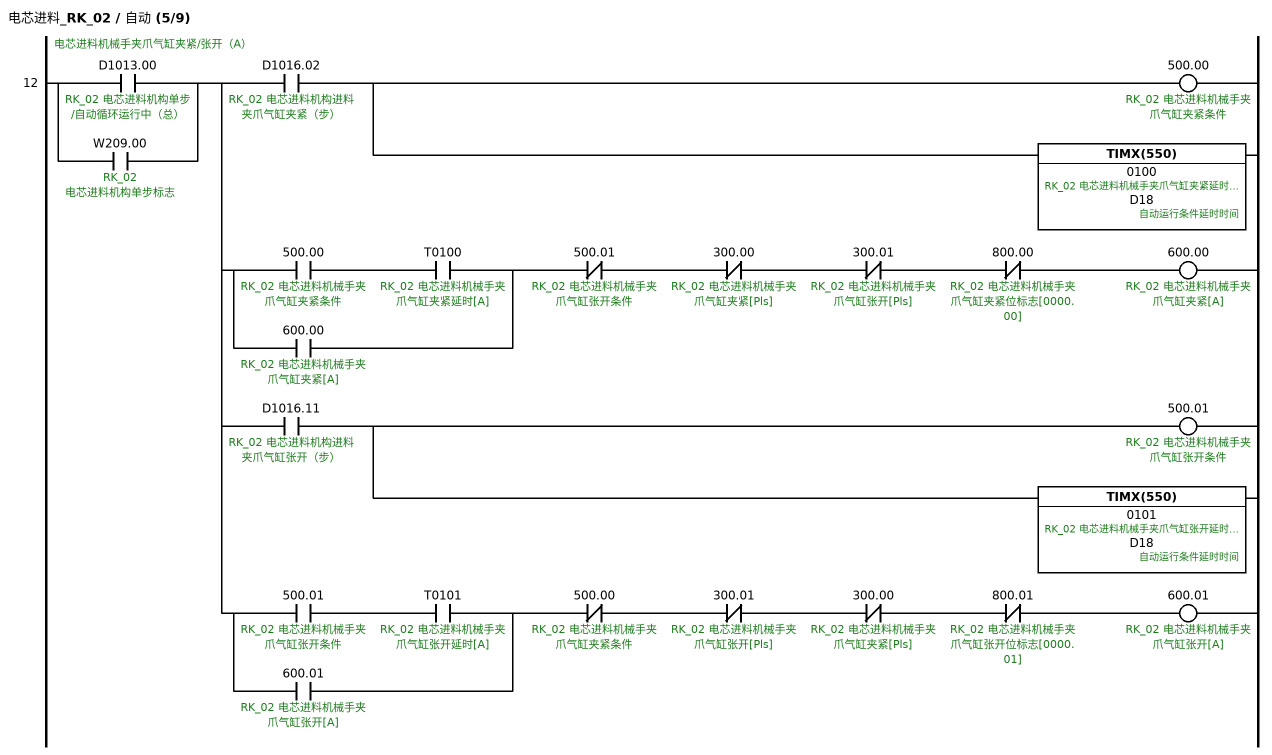
; [picture p360: 电芯进料_RK_02 / 自动, rungs 12-12]
; rung 12: 电芯进料机械手夹爪气缸夹紧/张开（A）
LD D1013.00  ; RK_02 电芯进料机构单步/自动循环运行中（总）
OR W209.00  ; RK_02  电芯进料机构单步标志
OUT TR0
AND D1016.02  ; RK_02 电芯进料机构进料夹爪气缸夹紧（步）
OUT 500.00  ; RK_02 电芯进料机械手夹爪气缸夹紧条件
TIMX(550) 0100 D18  ; 自动运行条件延时时间, RK_02 电芯进料机械手夹爪气缸夹紧延时[A]
LD TR0
LD 500.00  ; RK_02 电芯进料机械手夹爪气缸夹紧条件
AND T0100  ; RK_02 电芯进料机械手夹爪气缸夹紧延时[A]
OR 600.00  ; RK_02 电芯进料机械手夹爪气缸夹紧[A]
ANDLD
ANDNOT 500.01  ; RK_02 电芯进料机械手夹爪气缸张开条件
ANDNOT 300.00  ; RK_02 电芯进料机械手夹爪气缸夹紧[Pls]
ANDNOT 300.01  ; RK_02 电芯进料机械手夹爪气缸张开[Pls]
ANDNOT 800.00  ; RK_02 电芯进料机械手夹爪气缸夹紧位标志[0000.00]
OUT 600.00  ; RK_02 电芯进料机械手夹爪气缸夹紧[A]
LD TR0
AND D1016.11  ; RK_02 电芯进料机构进料夹爪气缸张开（步）
OUT 500.01  ; RK_02 电芯进料机械手夹爪气缸张开条件
TIMX(550) 0101 D18  ; 自动运行条件延时时间, RK_02 电芯进料机械手夹爪气缸张开延时[A]
LD TR0
LD 500.01  ; RK_02 电芯进料机械手夹爪气缸张开条件
AND T0101  ; RK_02 电芯进料机械手夹爪气缸张开延时[A]
OR 600.01  ; RK_02 电芯进料机械手夹爪气缸张开[A]
ANDLD
ANDNOT 500.00  ; RK_02 电芯进料机械手夹爪气缸夹紧条件
ANDNOT 300.01  ; RK_02 电芯进料机械手夹爪气缸张开[Pls]
ANDNOT 300.00  ; RK_02 电芯进料机械手夹爪气缸夹紧[Pls]
ANDNOT 800.01  ; RK_02 电芯进料机械手夹爪气缸张开位标志[0000.01]
OUT 600.01  ; RK_02 电芯进料机械手夹爪气缸张开[A]

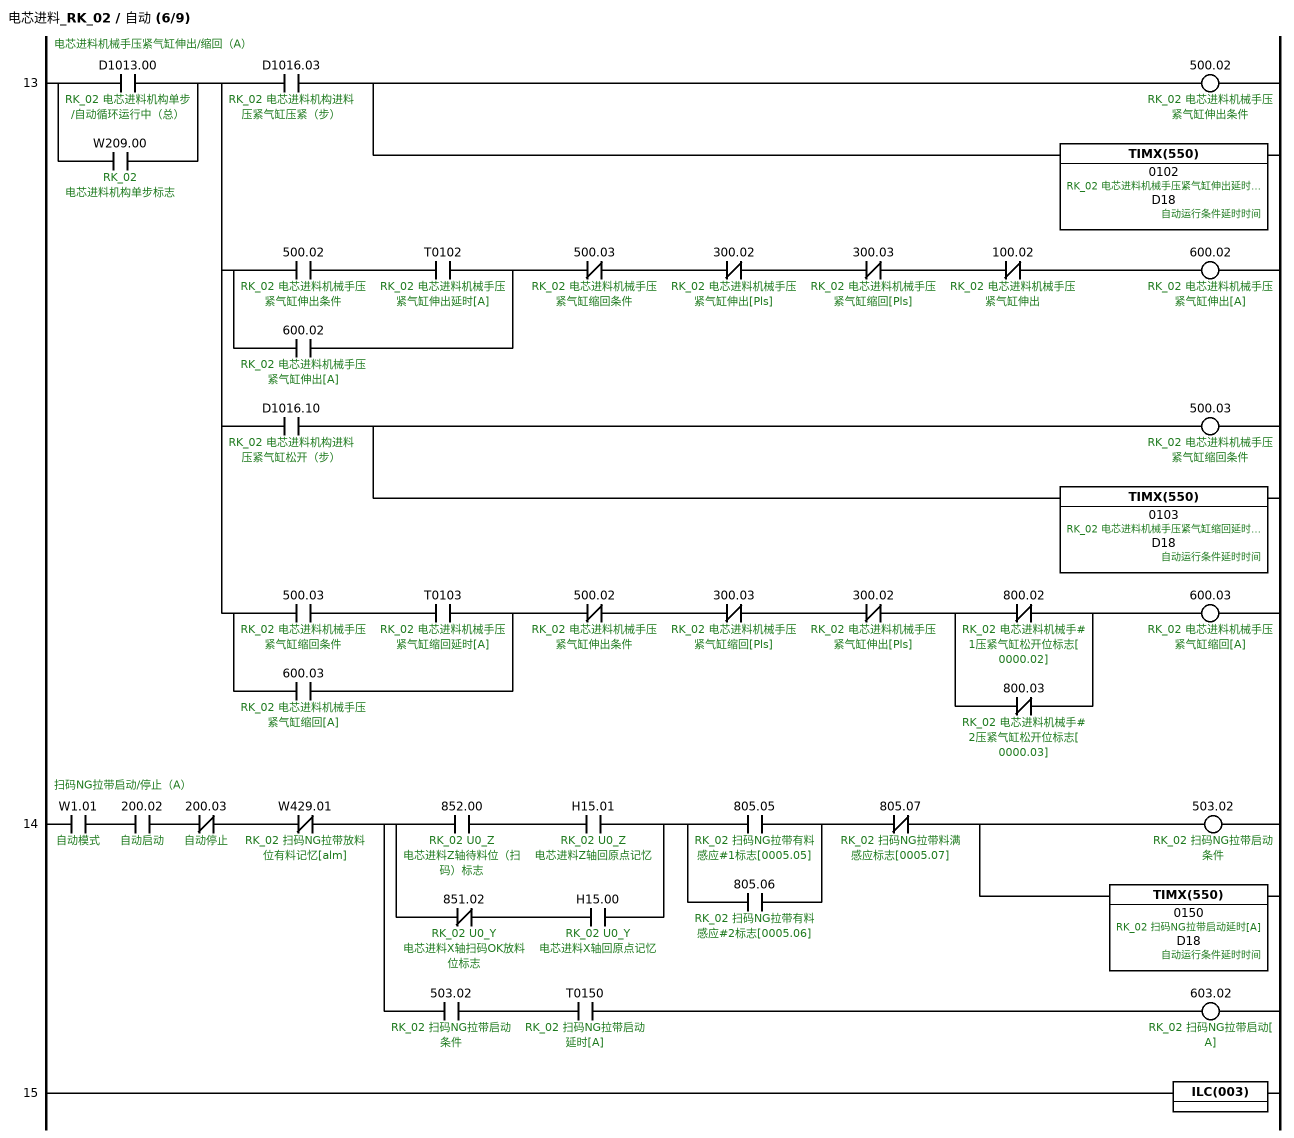
; rung 13: 电芯进料机械手压紧气缸伸出/缩回（A）
LD D1013.00  ; RK_02 电芯进料机构单步/自动循环运行中（总）
OR W209.00  ; RK_02  电芯进料机构单步标志
OUT TR0
AND D1016.03  ; RK_02 电芯进料机构进料压紧气缸压紧（步）
OUT 500.02  ; RK_02 电芯进料机械手压紧气缸伸出条件
TIMX(550) 0102 D18  ; 自动运行条件延时时间, RK_02 电芯进料机械手压紧气缸伸出延时[A]
LD TR0
LD 500.02  ; RK_02 电芯进料机械手压紧气缸伸出条件
AND T0102  ; RK_02 电芯进料机械手压紧气缸伸出延时[A]
OR 600.02  ; RK_02 电芯进料机械手压紧气缸伸出[A]
ANDLD
ANDNOT 500.03  ; RK_02 电芯进料机械手压紧气缸缩回条件
ANDNOT 300.02  ; RK_02 电芯进料机械手压紧气缸伸出[Pls]
ANDNOT 300.03  ; RK_02 电芯进料机械手压紧气缸缩回[Pls]
ANDNOT 100.02  ; RK_02 电芯进料机械手压紧气缸伸出
OUT 600.02  ; RK_02 电芯进料机械手压紧气缸伸出[A]
LD TR0
AND D1016.10  ; RK_02 电芯进料机构进料压紧气缸松开（步）
OUT 500.03  ; RK_02 电芯进料机械手压紧气缸缩回条件
TIMX(550) 0103 D18  ; 自动运行条件延时时间, RK_02 电芯进料机械手压紧气缸缩回延时[A]
LD TR0
LD 500.03  ; RK_02 电芯进料机械手压紧气缸缩回条件
AND T0103  ; RK_02 电芯进料机械手压紧气缸缩回延时[A]
OR 600.03  ; RK_02 电芯进料机械手压紧气缸缩回[A]
ANDLD
ANDNOT 500.02  ; RK_02 电芯进料机械手压紧气缸伸出条件
ANDNOT 300.03  ; RK_02 电芯进料机械手压紧气缸缩回[Pls]
ANDNOT 300.02  ; RK_02 电芯进料机械手压紧气缸伸出[Pls]
LDNOT 800.02  ; RK_02 电芯进料机械手#1压紧气缸松开位标志[0000.02]
ORNOT 800.03  ; RK_02 电芯进料机械手#2压紧气缸松开位标志[0000.03]
ANDLD
OUT 600.03  ; RK_02 电芯进料机械手压紧气缸缩回[A]
; rung 14: 扫码NG拉带启动/停止（A）
LD W1.01  ; 自动模式
AND 200.02  ; 自动启动
ANDNOT 200.03  ; 自动停止
ANDNOT W429.01  ; RK_02 扫码NG拉带放料位有料记忆[alm]
OUT TR0
LD 852.00  ; RK_02 U0_Z 电芯进料Z轴待料位（扫码）标志
AND H15.01  ; RK_02 U0_Z 电芯进料Z轴回原点记忆
LDNOT 851.02  ; RK_02 U0_Y 电芯进料X轴扫码OK放料位标志
AND H15.00  ; RK_02 U0_Y 电芯进料X轴回原点记忆
ORLD
ANDLD
LD 805.05  ; RK_02 扫码NG拉带有料感应#1标志[0005.05]
OR 805.06  ; RK_02 扫码NG拉带有料感应#2标志[0005.06]
ANDLD
ANDNOT 805.07  ; RK_02 扫码NG拉带料满感应标志[0005.07]
OUT 503.02  ; RK_02 扫码NG拉带启动条件
TIMX(550) 0150 D18  ; 自动运行条件延时时间, RK_02 扫码NG拉带启动延时[A]
LD TR0
AND 503.02  ; RK_02 扫码NG拉带启动条件
AND T0150  ; RK_02 扫码NG拉带启动延时[A]
OUT 603.02  ; RK_02 扫码NG拉带启动[A]
; rung 15
ILC(003)

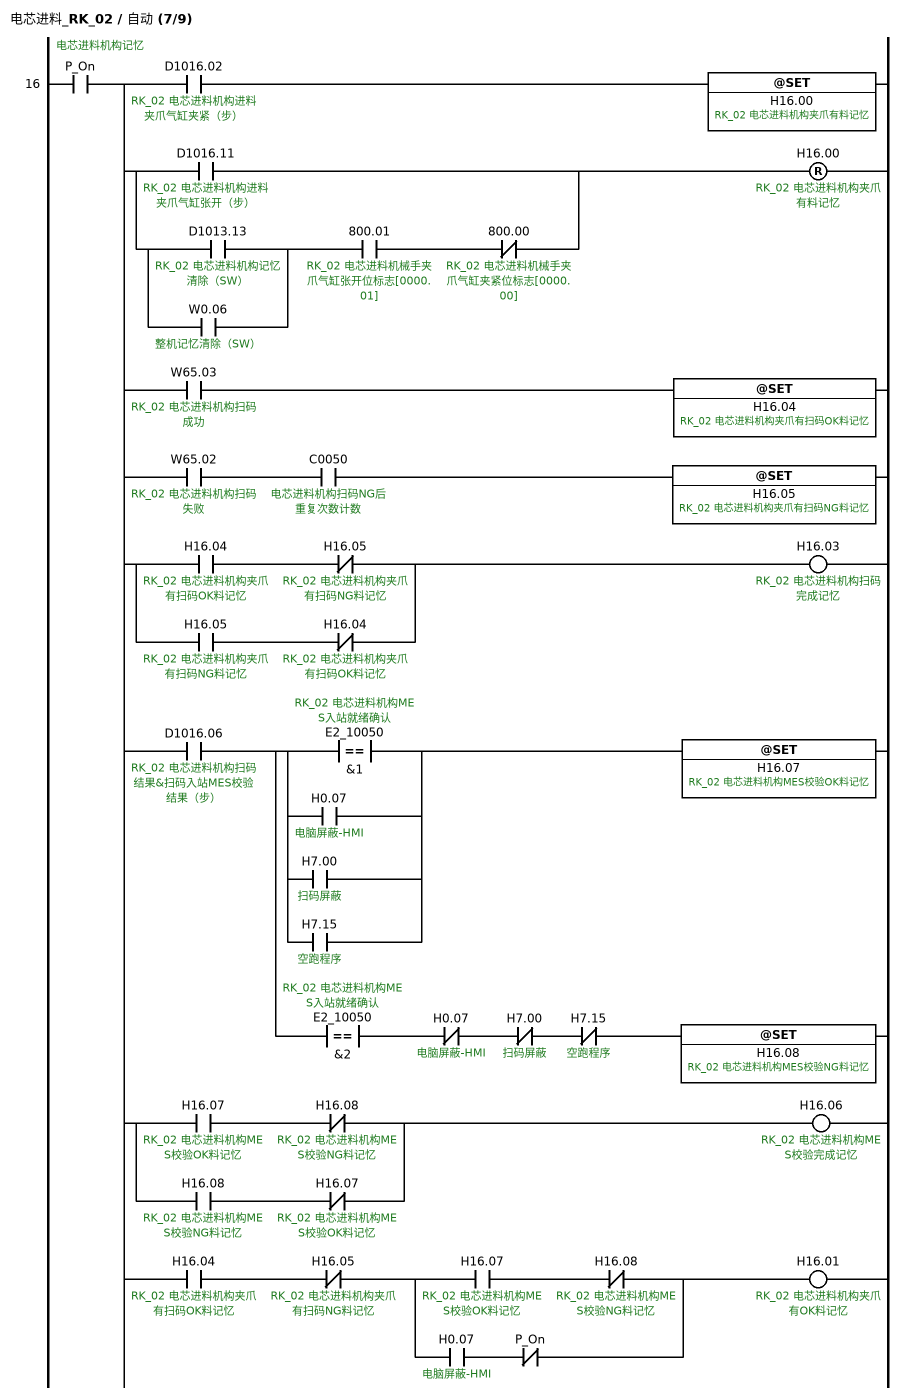

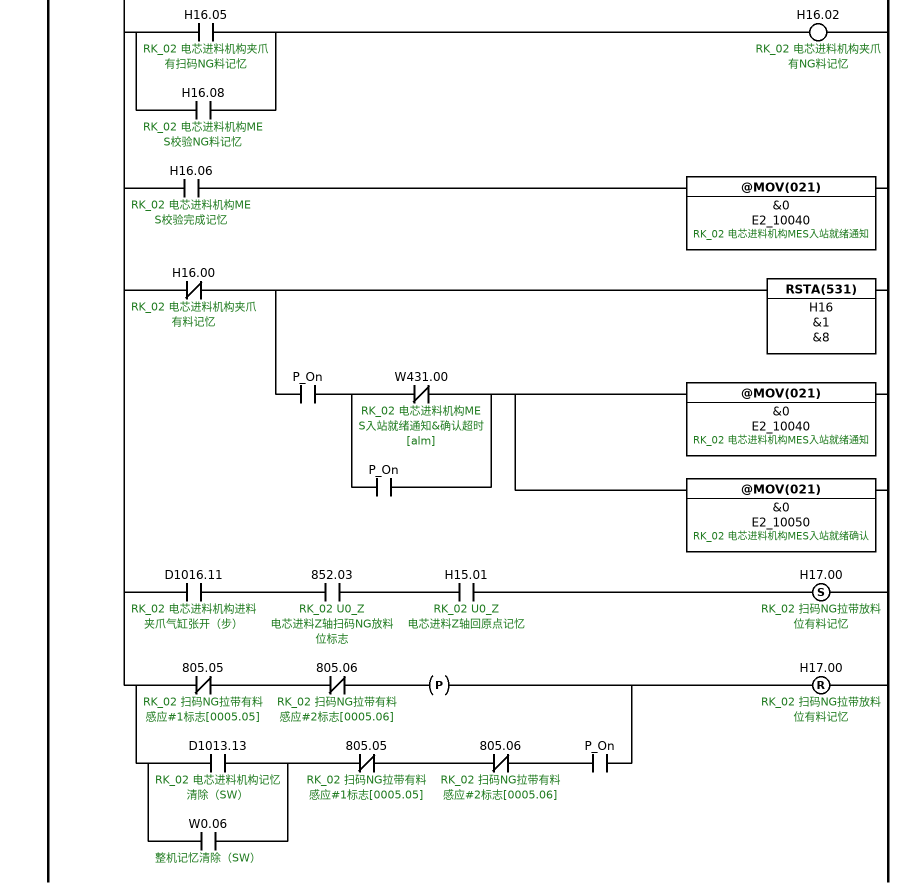
; rung 16: 电芯进料机构记忆
LD P_On
OUT TR0
AND D1016.02  ; RK_02 电芯进料机构进料夹爪气缸夹紧（步）
@SET H16.00  ; RK_02 电芯进料机构夹爪有料记忆
LD TR0
LD D1016.11  ; RK_02 电芯进料机构进料夹爪气缸张开（步）
LD D1013.13  ; RK_02 电芯进料机构记忆清除（SW）
OR W0.06  ; 整机记忆清除（SW）
AND 800.01  ; RK_02 电芯进料机械手夹爪气缸张开位标志[0000.01]
ANDNOT 800.00  ; RK_02 电芯进料机械手夹爪气缸夹紧位标志[0000.00]
ORLD
ANDLD
RSET H16.00  ; RK_02 电芯进料机构夹爪有料记忆
LD TR0
AND W65.03  ; RK_02 电芯进料机构扫码成功
@SET H16.04  ; RK_02 电芯进料机构夹爪有扫码OK料记忆
LD TR0
AND W65.02  ; RK_02 电芯进料机构扫码失败
AND C0050  ; 电芯进料机构扫码NG后重复次数计数
@SET H16.05  ; RK_02 电芯进料机构夹爪有扫码NG料记忆
LD TR0
LD H16.04  ; RK_02 电芯进料机构夹爪有扫码OK料记忆
ANDNOT H16.05  ; RK_02 电芯进料机构夹爪有扫码NG料记忆
LD H16.05  ; RK_02 电芯进料机构夹爪有扫码NG料记忆
ANDNOT H16.04  ; RK_02 电芯进料机构夹爪有扫码OK料记忆
ORLD
ANDLD
OUT H16.03  ; RK_02 电芯进料机构扫码完成记忆
LD TR0
AND D1016.06  ; RK_02 电芯进料机构扫码结果&扫码入站MES校验结果（步）
OUT TR1
LD=(300) E2_10050 &1  ; RK_02 电芯进料机构MES入站就绪确认  // 入站就绪确认=0：未确认，1：确认OK，2：确认NG
OR H0.07  ; 电脑屏蔽-HMI
OR H7.00  ; 扫码屏蔽
OR H7.15  ; 空跑程序
ANDLD
@SET H16.07  ; RK_02 电芯进料机构MES校验OK料记忆
LD TR1
AND=(300) E2_10050 &2  ; RK_02 电芯进料机构MES入站就绪确认  // 入站就绪确认=0：未确认，1：确认OK，2：确认NG
ANDNOT H0.07  ; 电脑屏蔽-HMI
ANDNOT H7.00  ; 扫码屏蔽
ANDNOT H7.15  ; 空跑程序
@SET H16.08  ; RK_02 电芯进料机构MES校验NG料记忆
LD TR0
LD H16.07  ; RK_02 电芯进料机构MES校验OK料记忆
ANDNOT H16.08  ; RK_02 电芯进料机构MES校验NG料记忆
LD H16.08  ; RK_02 电芯进料机构MES校验NG料记忆
ANDNOT H16.07  ; RK_02 电芯进料机构MES校验OK料记忆
ORLD
ANDLD
OUT H16.06  ; RK_02 电芯进料机构MES校验完成记忆
LD TR0
AND H16.04  ; RK_02 电芯进料机构夹爪有扫码OK料记忆
ANDNOT H16.05  ; RK_02 电芯进料机构夹爪有扫码NG料记忆
LD H16.07  ; RK_02 电芯进料机构MES校验OK料记忆
ANDNOT H16.08  ; RK_02 电芯进料机构MES校验NG料记忆
LD H0.07  ; 电脑屏蔽-HMI
ANDNOT P_On
ORLD
ANDLD
OUT H16.01  ; RK_02 电芯进料机构夹爪有OK料记忆
LD TR0
LD H16.05  ; RK_02 电芯进料机构夹爪有扫码NG料记忆
OR H16.08  ; RK_02 电芯进料机构MES校验NG料记忆
ANDLD
OUT H16.02  ; RK_02 电芯进料机构夹爪有NG料记忆
LD TR0
AND H16.06  ; RK_02 电芯进料机构MES校验完成记忆
@MOV(021) &0 E2_10040  ; RK_02 电芯进料机构MES入站就绪通知
LD TR0
ANDNOT H16.00  ; RK_02 电芯进料机构夹爪有料记忆
RSTA(531) H16 &1 &8
AND P_On
LDNOT W431.00  ; RK_02 电芯进料机构MES入站就绪通知&确认超时[alm]  // 工站夹爪没料且无MES入站就绪通知&确认报警条件下，RK_02 电芯进料机构MES入站就绪通知&确认才能清零
OR P_On
ANDLD
@MOV(021) &0 E2_10040  ; RK_02 电芯进料机构MES入站就绪通知
@MOV(021) &0 E2_10050  ; RK_02 电芯进料机构MES入站就绪确认
LD TR0
AND D1016.11  ; RK_02 电芯进料机构进料夹爪气缸张开（步）
AND 852.03  ; RK_02 U0_Z 电芯进料Z轴扫码NG放料位标志
AND H15.01  ; RK_02 U0_Z 电芯进料Z轴回原点记忆
SET H17.00  ; RK_02 扫码NG拉带放料位有料记忆
LD TR0
LDNOT 805.05  ; RK_02 扫码NG拉带有料感应#1标志[0005.05]
ANDNOT 805.06  ; RK_02 扫码NG拉带有料感应#2标志[0005.06]
UP(521)
LD D1013.13  ; RK_02 电芯进料机构记忆清除（SW）
OR W0.06  ; 整机记忆清除（SW）
ANDNOT 805.05  ; RK_02 扫码NG拉带有料感应#1标志[0005.05]
ANDNOT 805.06  ; RK_02 扫码NG拉带有料感应#2标志[0005.06]
AND P_On
ORLD
ANDLD
RSET H17.00  ; RK_02 扫码NG拉带放料位有料记忆

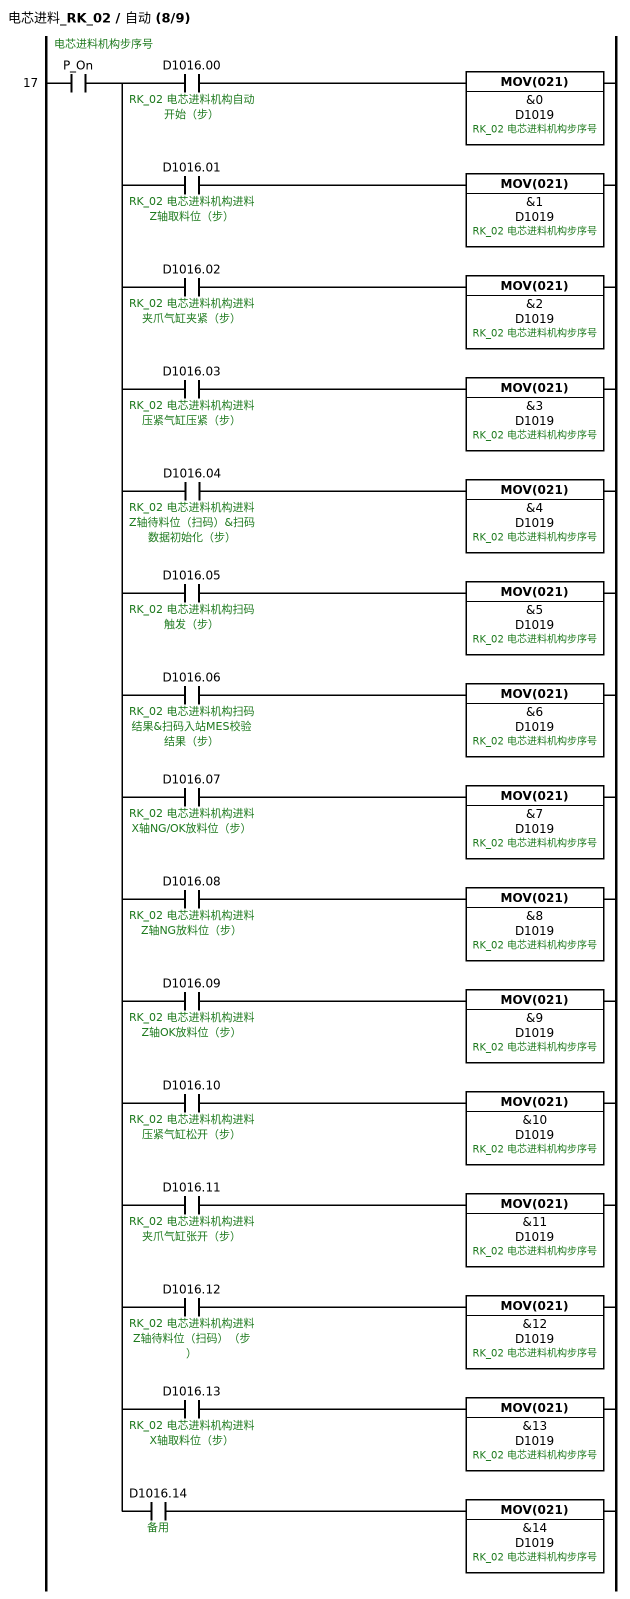
; rung 17: 电芯进料机构步序号
LD P_On
OUT TR0
AND D1016.00  ; RK_02 电芯进料机构自动开始（步）
MOV(021) &0 D1019  ; RK_02 电芯进料机构步序号
LD TR0
AND D1016.01  ; RK_02 电芯进料机构进料Z轴取料位（步）
MOV(021) &1 D1019  ; RK_02 电芯进料机构步序号
LD TR0
AND D1016.02  ; RK_02 电芯进料机构进料夹爪气缸夹紧（步）
MOV(021) &2 D1019  ; RK_02 电芯进料机构步序号
LD TR0
AND D1016.03  ; RK_02 电芯进料机构进料压紧气缸压紧（步）
MOV(021) &3 D1019  ; RK_02 电芯进料机构步序号
LD TR0
AND D1016.04  ; RK_02 电芯进料机构进料Z轴待料位（扫码）&扫码数据初始化（步）
MOV(021) &4 D1019  ; RK_02 电芯进料机构步序号
LD TR0
AND D1016.05  ; RK_02 电芯进料机构扫码触发（步）
MOV(021) &5 D1019  ; RK_02 电芯进料机构步序号
LD TR0
AND D1016.06  ; RK_02 电芯进料机构扫码结果&扫码入站MES校验结果（步）
MOV(021) &6 D1019  ; RK_02 电芯进料机构步序号
LD TR0
AND D1016.07  ; RK_02 电芯进料机构进料X轴NG/OK放料位（步）
MOV(021) &7 D1019  ; RK_02 电芯进料机构步序号
LD TR0
AND D1016.08  ; RK_02 电芯进料机构进料Z轴NG放料位（步）
MOV(021) &8 D1019  ; RK_02 电芯进料机构步序号
LD TR0
AND D1016.09  ; RK_02 电芯进料机构进料Z轴OK放料位（步）
MOV(021) &9 D1019  ; RK_02 电芯进料机构步序号
LD TR0
AND D1016.10  ; RK_02 电芯进料机构进料压紧气缸松开（步）
MOV(021) &10 D1019  ; RK_02 电芯进料机构步序号
LD TR0
AND D1016.11  ; RK_02 电芯进料机构进料夹爪气缸张开（步）
MOV(021) &11 D1019  ; RK_02 电芯进料机构步序号
LD TR0
AND D1016.12  ; RK_02 电芯进料机构进料Z轴待料位（扫码）（步）
MOV(021) &12 D1019  ; RK_02 电芯进料机构步序号
LD TR0
AND D1016.13  ; RK_02 电芯进料机构进料X轴取料位（步）
MOV(021) &13 D1019  ; RK_02 电芯进料机构步序号
LD TR0
AND D1016.14  ; 备用
MOV(021) &14 D1019  ; RK_02 电芯进料机构步序号

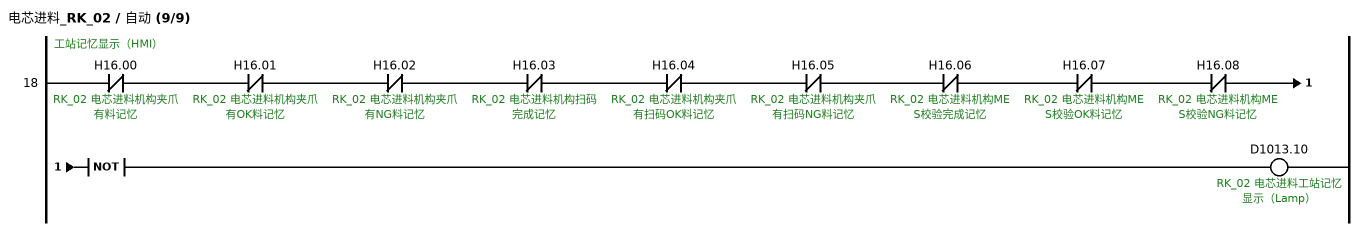
; rung 18: 工站记忆显示（HMI）
LDNOT H16.00  ; RK_02 电芯进料机构夹爪有料记忆
ANDNOT H16.01  ; RK_02 电芯进料机构夹爪有OK料记忆
ANDNOT H16.02  ; RK_02 电芯进料机构夹爪有NG料记忆
ANDNOT H16.03  ; RK_02 电芯进料机构扫码完成记忆
ANDNOT H16.04  ; RK_02 电芯进料机构夹爪有扫码OK料记忆
ANDNOT H16.05  ; RK_02 电芯进料机构夹爪有扫码NG料记忆
ANDNOT H16.06  ; RK_02 电芯进料机构MES校验完成记忆
ANDNOT H16.07  ; RK_02 电芯进料机构MES校验OK料记忆
ANDNOT H16.08  ; RK_02 电芯进料机构MES校验NG料记忆
NOT(520)
OUT D1013.10  ; RK_02 电芯进料工站记忆显示（Lamp）

### Section 复位

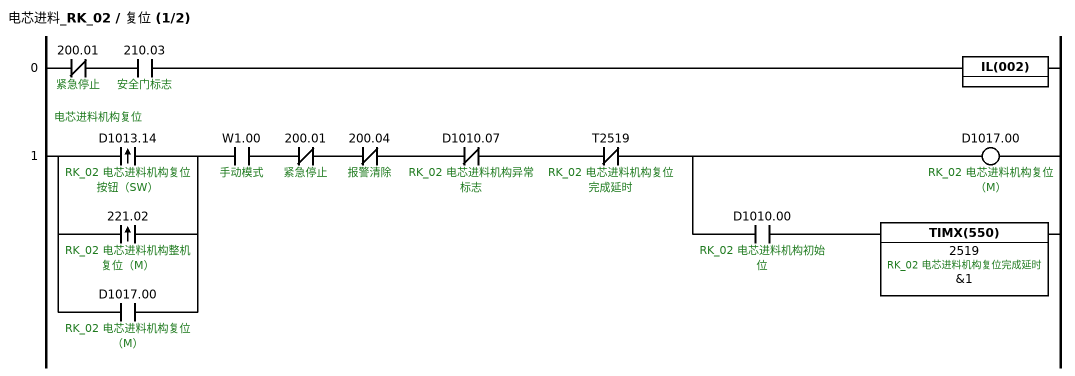
; rung 0
LDNOT 200.01  ; 紧急停止
AND 210.03  ; 安全门标志
IL(002)
; rung 1: 电芯进料机构复位
@LD D1013.14  ; RK_02 电芯进料机构复位按钮（SW）
@OR 221.02  ; RK_02 电芯进料机构整机复位（M）
OR D1017.00  ; RK_02 电芯进料机构复位（M）
AND W1.00  ; 手动模式
ANDNOT 200.01  ; 紧急停止
ANDNOT 200.04  ; 报警清除
ANDNOT D1010.07  ; RK_02 电芯进料机构异常标志
ANDNOT T2519  ; RK_02 电芯进料机构复位完成延时
OUT D1017.00  ; RK_02 电芯进料机构复位（M）
AND D1010.00  ; RK_02 电芯进料机构初始位
TIMX(550) 2519 &1  ; RK_02 电芯进料机构复位完成延时

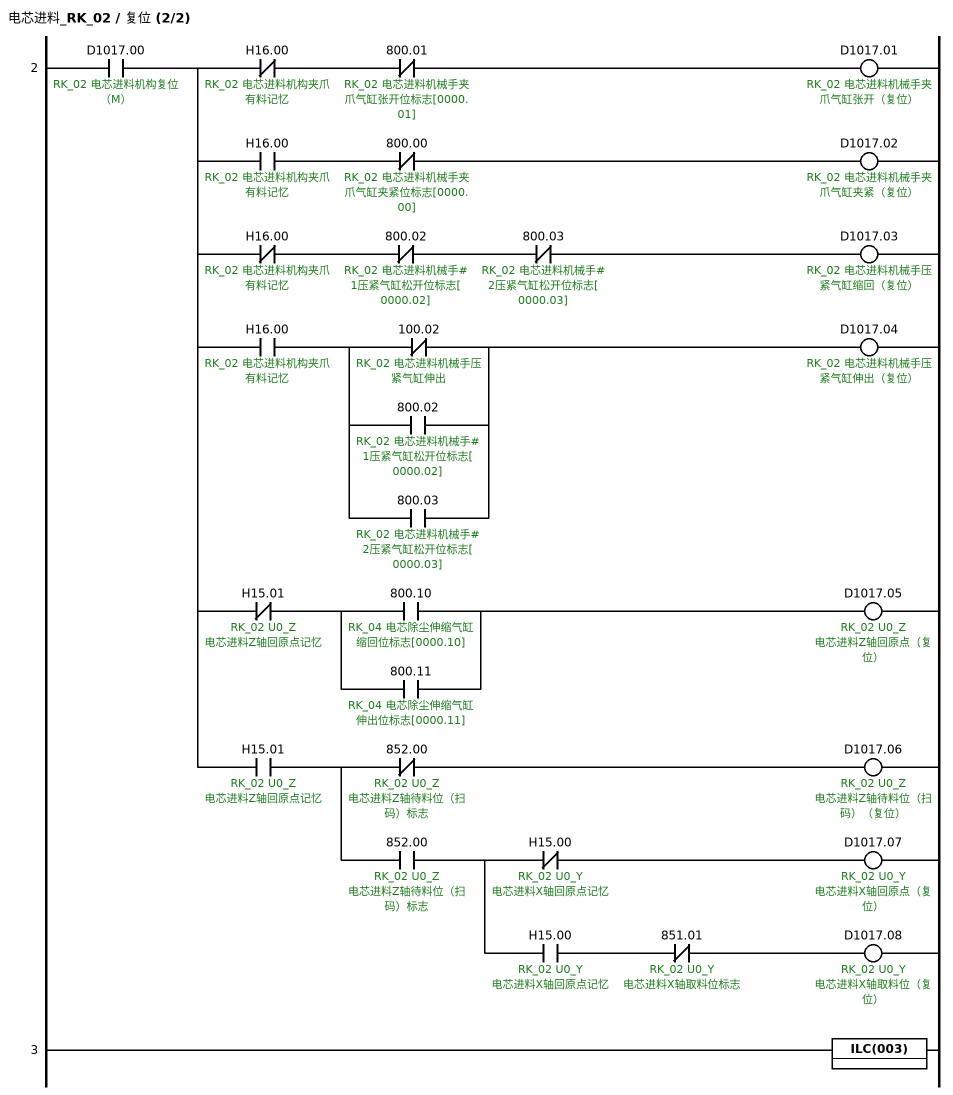
; rung 2
LD D1017.00  ; RK_02 电芯进料机构复位（M）
OUT TR0
ANDNOT H16.00  ; RK_02 电芯进料机构夹爪有料记忆
ANDNOT 800.01  ; RK_02 电芯进料机械手夹爪气缸张开位标志[0000.01]
OUT D1017.01  ; RK_02 电芯进料机械手夹爪气缸张开（复位）
LD TR0
AND H16.00  ; RK_02 电芯进料机构夹爪有料记忆
ANDNOT 800.00  ; RK_02 电芯进料机械手夹爪气缸夹紧位标志[0000.00]
OUT D1017.02  ; RK_02 电芯进料机械手夹爪气缸夹紧（复位）
LD TR0
ANDNOT H16.00  ; RK_02 电芯进料机构夹爪有料记忆
ANDNOT 800.02  ; RK_02 电芯进料机械手#1压紧气缸松开位标志[0000.02]
ANDNOT 800.03  ; RK_02 电芯进料机械手#2压紧气缸松开位标志[0000.03]
OUT D1017.03  ; RK_02 电芯进料机械手压紧气缸缩回（复位）
LD TR0
AND H16.00  ; RK_02 电芯进料机构夹爪有料记忆
LDNOT 100.02  ; RK_02 电芯进料机械手压紧气缸伸出
OR 800.02  ; RK_02 电芯进料机械手#1压紧气缸松开位标志[0000.02]
OR 800.03  ; RK_02 电芯进料机械手#2压紧气缸松开位标志[0000.03]
ANDLD
OUT D1017.04  ; RK_02 电芯进料机械手压紧气缸伸出（复位）
LD TR0
ANDNOT H15.01  ; RK_02 U0_Z 电芯进料Z轴回原点记忆
LD 800.10  ; RK_04 电芯除尘伸缩气缸缩回位标志[0000.10]
OR 800.11  ; RK_04 电芯除尘伸缩气缸伸出位标志[0000.11]
ANDLD
OUT D1017.05  ; RK_02 U0_Z 电芯进料Z轴回原点（复位）
LD TR0
AND H15.01  ; RK_02 U0_Z 电芯进料Z轴回原点记忆
OUT TR0
ANDNOT 852.00  ; RK_02 U0_Z 电芯进料Z轴待料位（扫码）标志
OUT D1017.06  ; RK_02 U0_Z 电芯进料Z轴待料位（扫码）（复位）
LD TR0
AND 852.00  ; RK_02 U0_Z 电芯进料Z轴待料位（扫码）标志
OUT TR0
ANDNOT H15.00  ; RK_02 U0_Y 电芯进料X轴回原点记忆
OUT D1017.07  ; RK_02 U0_Y 电芯进料X轴回原点（复位）
LD TR0
AND H15.00  ; RK_02 U0_Y 电芯进料X轴回原点记忆
ANDNOT 851.01  ; RK_02 U0_Y 电芯进料X轴取料位标志
OUT D1017.08  ; RK_02 U0_Y 电芯进料X轴取料位（复位）
; rung 3
ILC(003)

### Section 指示灯

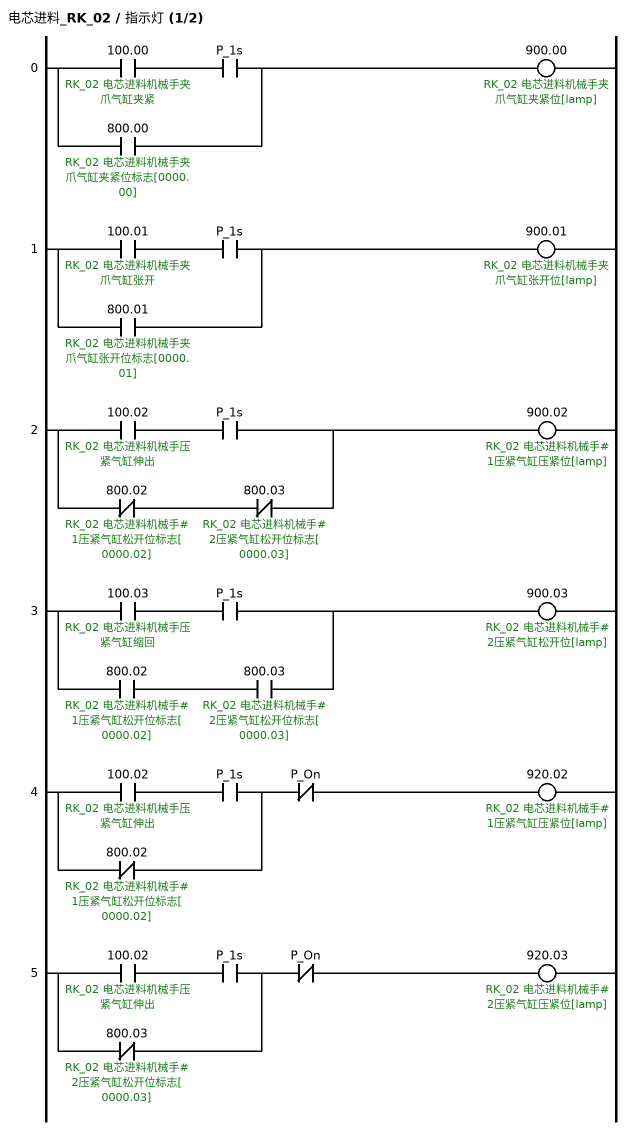
; rung 0
LD 100.00  ; RK_02 电芯进料机械手夹爪气缸夹紧
AND P_1s
OR 800.00  ; RK_02 电芯进料机械手夹爪气缸夹紧位标志[0000.00]
OUT 900.00  ; RK_02 电芯进料机械手夹爪气缸夹紧位[lamp]
; rung 1
LD 100.01  ; RK_02 电芯进料机械手夹爪气缸张开
AND P_1s
OR 800.01  ; RK_02 电芯进料机械手夹爪气缸张开位标志[0000.01]
OUT 900.01  ; RK_02 电芯进料机械手夹爪气缸张开位[lamp]
; rung 2
LD 100.02  ; RK_02 电芯进料机械手压紧气缸伸出
AND P_1s
LDNOT 800.02  ; RK_02 电芯进料机械手#1压紧气缸松开位标志[0000.02]
ANDNOT 800.03  ; RK_02 电芯进料机械手#2压紧气缸松开位标志[0000.03]
ORLD
OUT 900.02  ; RK_02 电芯进料机械手#1压紧气缸压紧位[lamp]
; rung 3
LD 100.03  ; RK_02 电芯进料机械手压紧气缸缩回
AND P_1s
LD 800.02  ; RK_02 电芯进料机械手#1压紧气缸松开位标志[0000.02]
AND 800.03  ; RK_02 电芯进料机械手#2压紧气缸松开位标志[0000.03]
ORLD
OUT 900.03  ; RK_02 电芯进料机械手#2压紧气缸松开位[lamp]
; rung 4
LD 100.02  ; RK_02 电芯进料机械手压紧气缸伸出
AND P_1s
ORNOT 800.02  ; RK_02 电芯进料机械手#1压紧气缸松开位标志[0000.02]
ANDNOT P_On
OUT 920.02  ; RK_02 电芯进料机械手#1压紧气缸压紧位[lamp]
; rung 5
LD 100.02  ; RK_02 电芯进料机械手压紧气缸伸出
AND P_1s
ORNOT 800.03  ; RK_02 电芯进料机械手#2压紧气缸松开位标志[0000.03]
ANDNOT P_On
OUT 920.03  ; RK_02 电芯进料机械手#2压紧气缸压紧位[lamp]

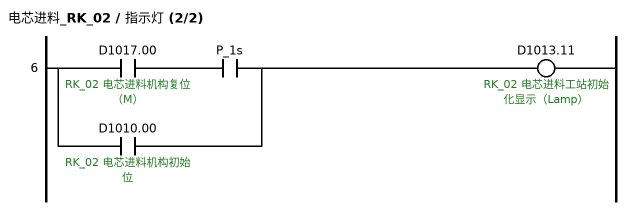
; rung 6
LD D1017.00  ; RK_02 电芯进料机构复位（M）
AND P_1s
OR D1010.00  ; RK_02 电芯进料机构初始位
OUT D1013.11  ; RK_02 电芯进料工站初始化显示（Lamp）

### Section 外部输出

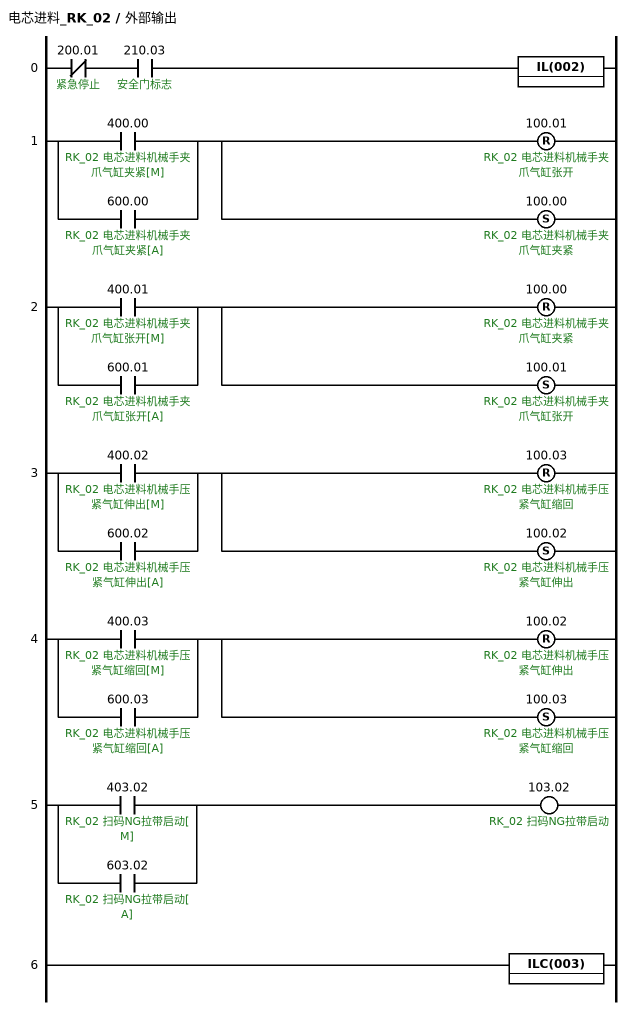
; rung 0
LDNOT 200.01  ; 紧急停止
AND 210.03  ; 安全门标志
IL(002)
; rung 1
LD 400.00  ; RK_02 电芯进料机械手夹爪气缸夹紧[M]
OR 600.00  ; RK_02 电芯进料机械手夹爪气缸夹紧[A]
RSET 100.01  ; RK_02 电芯进料机械手夹爪气缸张开
SET 100.00  ; RK_02 电芯进料机械手夹爪气缸夹紧
; rung 2
LD 400.01  ; RK_02 电芯进料机械手夹爪气缸张开[M]
OR 600.01  ; RK_02 电芯进料机械手夹爪气缸张开[A]
RSET 100.00  ; RK_02 电芯进料机械手夹爪气缸夹紧
SET 100.01  ; RK_02 电芯进料机械手夹爪气缸张开
; rung 3
LD 400.02  ; RK_02 电芯进料机械手压紧气缸伸出[M]
OR 600.02  ; RK_02 电芯进料机械手压紧气缸伸出[A]
RSET 100.03  ; RK_02 电芯进料机械手压紧气缸缩回
SET 100.02  ; RK_02 电芯进料机械手压紧气缸伸出
; rung 4
LD 400.03  ; RK_02 电芯进料机械手压紧气缸缩回[M]
OR 600.03  ; RK_02 电芯进料机械手压紧气缸缩回[A]
RSET 100.02  ; RK_02 电芯进料机械手压紧气缸伸出
SET 100.03  ; RK_02 电芯进料机械手压紧气缸缩回
; rung 5
LD 403.02  ; RK_02 扫码NG拉带启动[M]
OR 603.02  ; RK_02 扫码NG拉带启动[A]
OUT 103.02  ; RK_02 扫码NG拉带启动
; rung 6
ILC(003)

### Section END
; rung 0
END(001)

## Program 电芯上料_RK_03 (cyclic task 3)

### Section Main

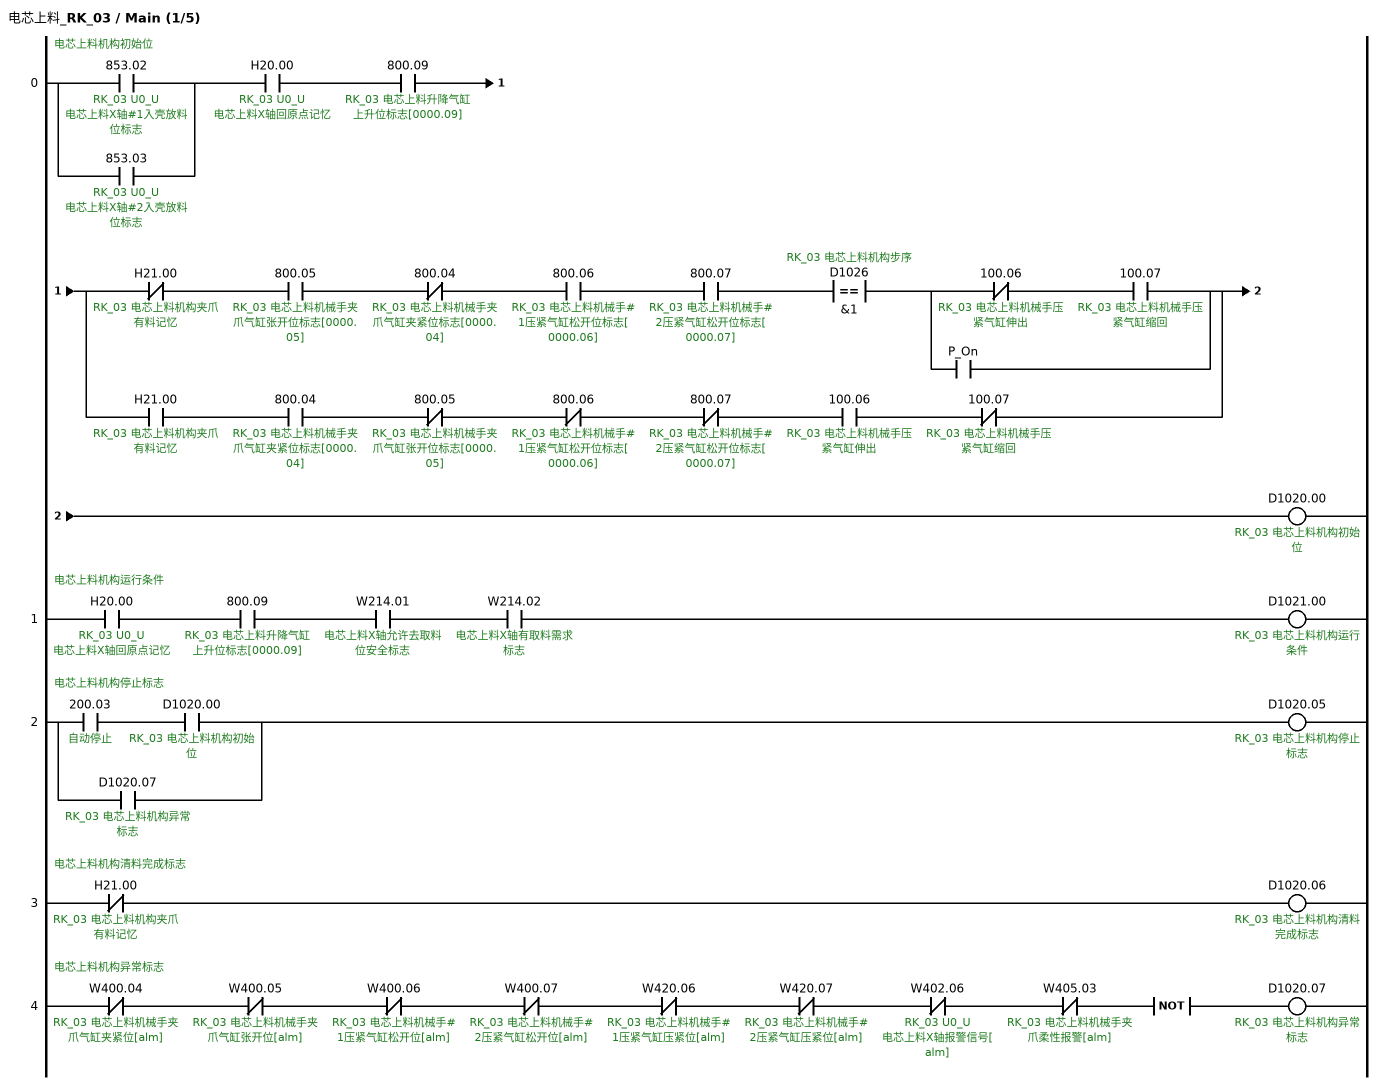
; rung 0: 电芯上料机构初始位
LD 853.02  ; RK_03 U0_U 电芯上料X轴#1入壳放料位标志
OR 853.03  ; RK_03 U0_U 电芯上料X轴#2入壳放料位标志
AND H20.00  ; RK_03 U0_U 电芯上料X轴回原点记忆
AND 800.09  ; RK_03 电芯上料升降气缸上升位标志[0000.09]
LDNOT H21.00  ; RK_03 电芯上料机构夹爪有料记忆
AND 800.05  ; RK_03 电芯上料机械手夹爪气缸张开位标志[0000.05]
ANDNOT 800.04  ; RK_03 电芯上料机械手夹爪气缸夹紧位标志[0000.04]
AND 800.06  ; RK_03 电芯上料机械手#1压紧气缸松开位标志[0000.06]
AND 800.07  ; RK_03 电芯上料机械手#2压紧气缸松开位标志[0000.07]
AND=(300) D1026 &1  ; RK_03 电芯上料机构步序
LDNOT 100.06  ; RK_03 电芯上料机械手压紧气缸伸出
AND 100.07  ; RK_03 电芯上料机械手压紧气缸缩回
OR P_On
ANDLD
LD H21.00  ; RK_03 电芯上料机构夹爪有料记忆
AND 800.04  ; RK_03 电芯上料机械手夹爪气缸夹紧位标志[0000.04]
ANDNOT 800.05  ; RK_03 电芯上料机械手夹爪气缸张开位标志[0000.05]
ANDNOT 800.06  ; RK_03 电芯上料机械手#1压紧气缸松开位标志[0000.06]
ANDNOT 800.07  ; RK_03 电芯上料机械手#2压紧气缸松开位标志[0000.07]
AND 100.06  ; RK_03 电芯上料机械手压紧气缸伸出
ANDNOT 100.07  ; RK_03 电芯上料机械手压紧气缸缩回
ORLD
ANDLD
OUT D1020.00  ; RK_03 电芯上料机构初始位
; rung 1: 电芯上料机构运行条件
LD H20.00  ; RK_03 U0_U 电芯上料X轴回原点记忆
AND 800.09  ; RK_03 电芯上料升降气缸上升位标志[0000.09]
AND W214.01  ; 电芯上料X轴允许去取料位安全标志
AND W214.02  ; 电芯上料X轴有取料需求标志
OUT D1021.00  ; RK_03 电芯上料机构运行条件
; rung 2: 电芯上料机构停止标志
LD 200.03  ; 自动停止
AND D1020.00  ; RK_03 电芯上料机构初始位
OR D1020.07  ; RK_03 电芯上料机构异常标志
OUT D1020.05  ; RK_03 电芯上料机构停止标志
; rung 3: 电芯上料机构清料完成标志
LDNOT H21.00  ; RK_03 电芯上料机构夹爪有料记忆
OUT D1020.06  ; RK_03 电芯上料机构清料完成标志
; rung 4: 电芯上料机构异常标志
LDNOT W400.04  ; RK_03 电芯上料机械手夹爪气缸夹紧位[alm]
ANDNOT W400.05  ; RK_03 电芯上料机械手夹爪气缸张开位[alm]
ANDNOT W400.06  ; RK_03 电芯上料机械手#1压紧气缸松开位[alm]
ANDNOT W400.07  ; RK_03 电芯上料机械手#2压紧气缸松开位[alm]
ANDNOT W420.06  ; RK_03 电芯上料机械手#1压紧气缸压紧位[alm]
ANDNOT W420.07  ; RK_03 电芯上料机械手#2压紧气缸压紧位[alm]
ANDNOT W402.06  ; RK_03 U0_U 电芯上料X轴报警信号[alm]
ANDNOT W405.03  ; RK_03 电芯上料机械手夹爪柔性报警[alm]
NOT(520)
OUT D1020.07  ; RK_03 电芯上料机构异常标志

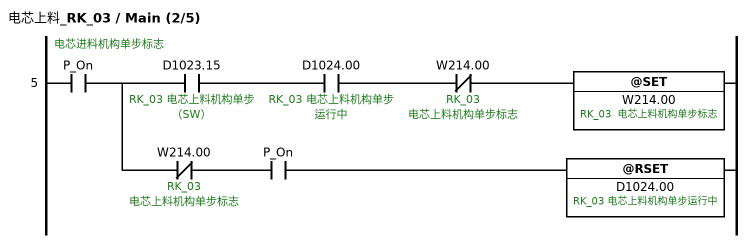
; rung 5: 电芯进料机构单步标志
LD P_On
OUT TR0
AND D1023.15  ; RK_03 电芯上料机构单步（SW）
AND D1024.00  ; RK_03 电芯上料机构单步运行中
ANDNOT W214.00  ; RK_03  电芯上料机构单步标志
@SET W214.00  ; RK_03  电芯上料机构单步标志
LD TR0
ANDNOT W214.00  ; RK_03  电芯上料机构单步标志
AND P_On
@RSET D1024.00  ; RK_03 电芯上料机构单步运行中

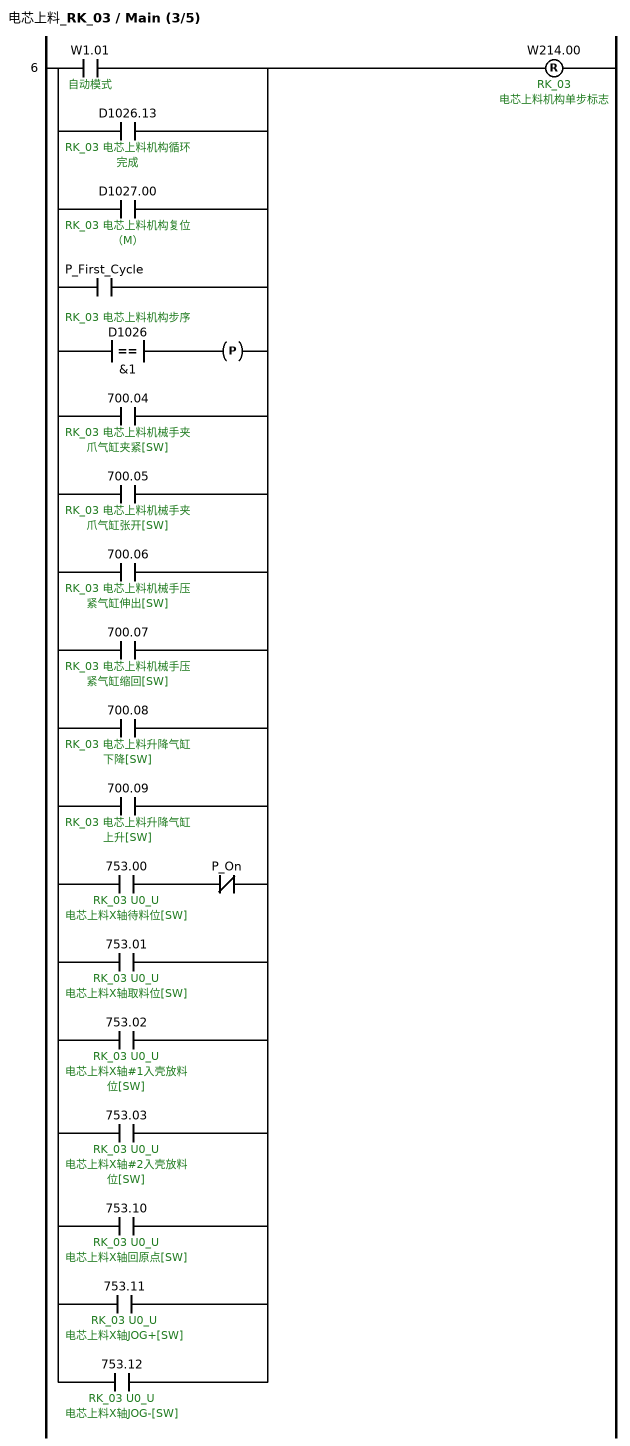
; rung 6
LD W1.01  ; 自动模式
OR D1026.13  ; RK_03 电芯上料机构循环完成
OR D1027.00  ; RK_03 电芯上料机构复位（M）
OR P_First_Cycle
LD=(300) D1026 &1  ; RK_03 电芯上料机构步序
UP(521)
ORLD
OR 700.04  ; RK_03 电芯上料机械手夹爪气缸夹紧[SW]
OR 700.05  ; RK_03 电芯上料机械手夹爪气缸张开[SW]
OR 700.06  ; RK_03 电芯上料机械手压紧气缸伸出[SW]
OR 700.07  ; RK_03 电芯上料机械手压紧气缸缩回[SW]
OR 700.08  ; RK_03 电芯上料升降气缸下降[SW]
OR 700.09  ; RK_03 电芯上料升降气缸上升[SW]
LD 753.00  ; RK_03 U0_U 电芯上料X轴待料位[SW]
ANDNOT P_On
ORLD
OR 753.01  ; RK_03 U0_U 电芯上料X轴取料位[SW]
OR 753.02  ; RK_03 U0_U 电芯上料X轴#1入壳放料位[SW]
OR 753.03  ; RK_03 U0_U 电芯上料X轴#2入壳放料位[SW]
OR 753.10  ; RK_03 U0_U 电芯上料X轴回原点[SW]
OR 753.11  ; RK_03 U0_U 电芯上料X轴JOG+[SW]
OR 753.12  ; RK_03 U0_U 电芯上料X轴JOG-[SW]
RSET W214.00  ; RK_03  电芯上料机构单步标志

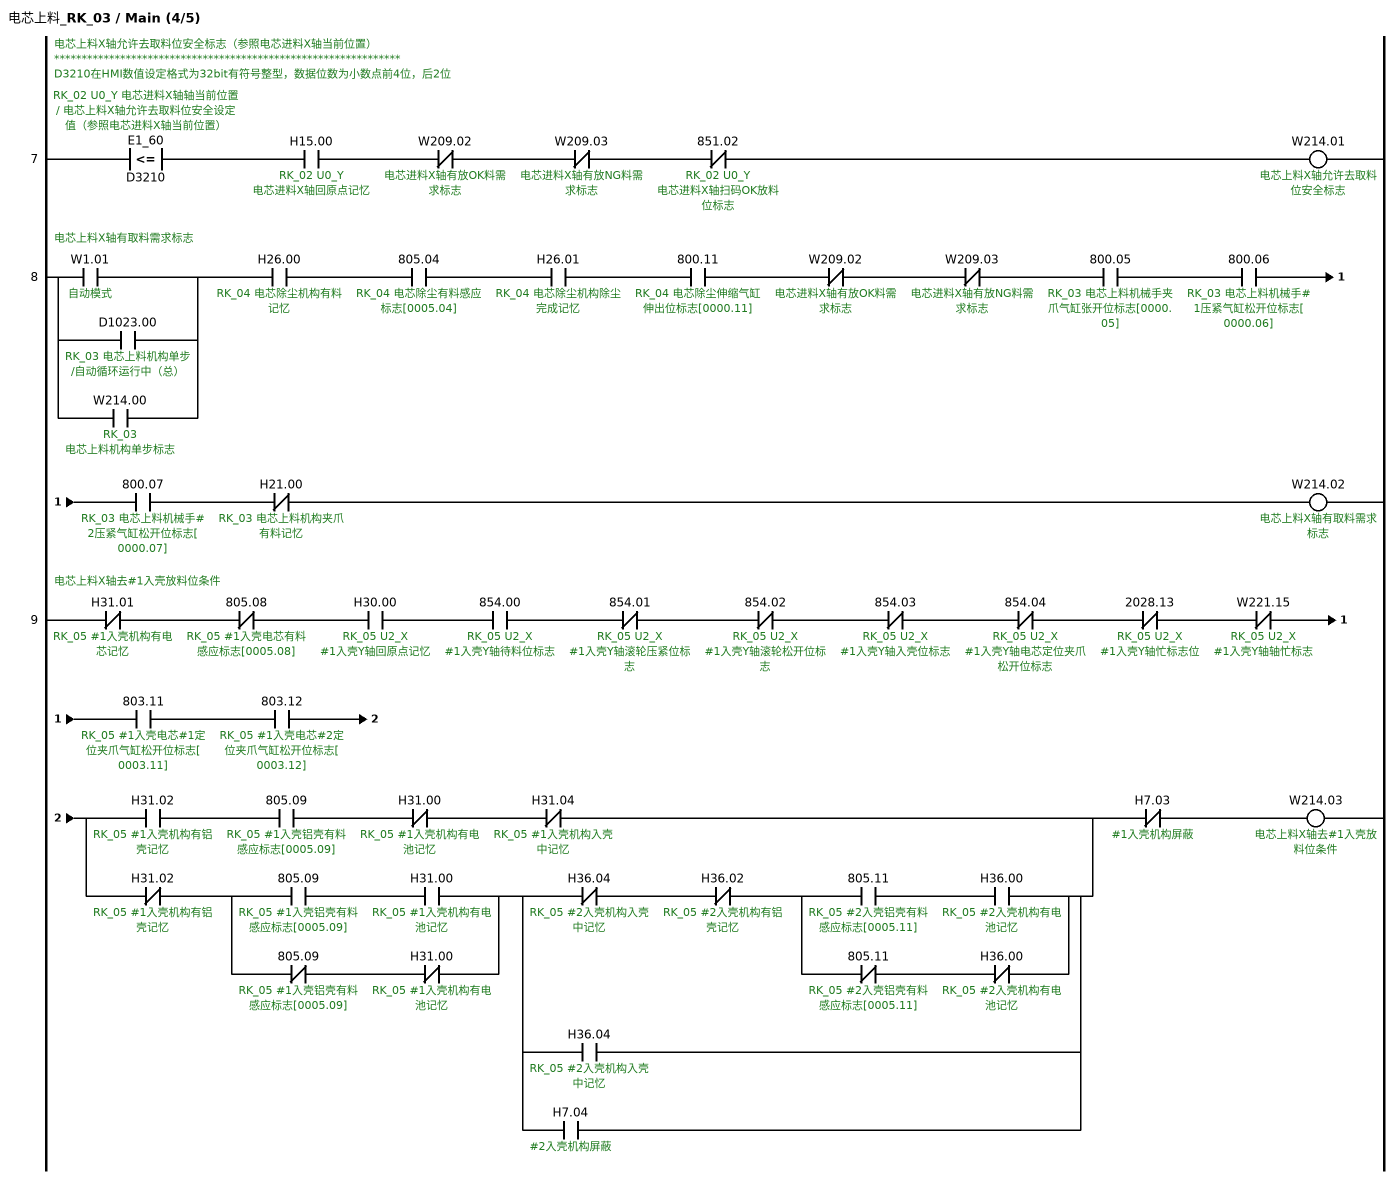
; rung 7: 电芯上料X轴允许去取料位安全标志（参照电芯进料X轴当前位置） / *************************************************************** / D3210在HMI数值设定格式为32bit有符号整型，数据位数为小数点前4位，后2位
LD<=SL(318) E1_60 D3210  ; RK_02 U0_Y 电芯进料X轴轴当前位置, 电芯上料X轴允许去取料位安全设定值（参照电芯进料X轴当前位置）
AND H15.00  ; RK_02 U0_Y 电芯进料X轴回原点记忆
ANDNOT W209.02  ; 电芯进料X轴有放OK料需求标志
ANDNOT W209.03  ; 电芯进料X轴有放NG料需求标志
ANDNOT 851.02  ; RK_02 U0_Y 电芯进料X轴扫码OK放料位标志
OUT W214.01  ; 电芯上料X轴允许去取料位安全标志
; rung 8: 电芯上料X轴有取料需求标志
LD W1.01  ; 自动模式
OR D1023.00  ; RK_03 电芯上料机构单步/自动循环运行中（总）
OR W214.00  ; RK_03  电芯上料机构单步标志
AND H26.00  ; RK_04 电芯除尘机构有料记忆
AND 805.04  ; RK_04 电芯除尘有料感应标志[0005.04]
AND H26.01  ; RK_04 电芯除尘机构除尘完成记忆
AND 800.11  ; RK_04 电芯除尘伸缩气缸伸出位标志[0000.11]
ANDNOT W209.02  ; 电芯进料X轴有放OK料需求标志
ANDNOT W209.03  ; 电芯进料X轴有放NG料需求标志
AND 800.05  ; RK_03 电芯上料机械手夹爪气缸张开位标志[0000.05]
AND 800.06  ; RK_03 电芯上料机械手#1压紧气缸松开位标志[0000.06]
AND 800.07  ; RK_03 电芯上料机械手#2压紧气缸松开位标志[0000.07]
ANDNOT H21.00  ; RK_03 电芯上料机构夹爪有料记忆
OUT W214.02  ; 电芯上料X轴有取料需求标志
; rung 9: 电芯上料X轴去#1入壳放料位条件
LDNOT H31.01  ; RK_05 #1入壳机构有电芯记忆
ANDNOT 805.08  ; RK_05 #1入壳电芯有料感应标志[0005.08]
AND H30.00  ; RK_05 U2_X #1入壳Y轴回原点记忆
AND 854.00  ; RK_05 U2_X #1入壳Y轴待料位标志
ANDNOT 854.01  ; RK_05 U2_X #1入壳Y轴滚轮压紧位标志
ANDNOT 854.02  ; RK_05 U2_X #1入壳Y轴滚轮松开位标志
ANDNOT 854.03  ; RK_05 U2_X #1入壳Y轴入壳位标志
ANDNOT 854.04  ; RK_05 U2_X #1入壳Y轴电芯定位夹爪松开位标志
ANDNOT 2028.13  ; RK_05 U2_X #1入壳Y轴忙标志位
ANDNOT W221.15  ; RK_05 U2_X #1入壳Y轴轴忙标志
AND 803.11  ; RK_05 #1入壳电芯#1定位夹爪气缸松开位标志[0003.11]
AND 803.12  ; RK_05 #1入壳电芯#2定位夹爪气缸松开位标志[0003.12]
LD H31.02  ; RK_05 #1入壳机构有铝壳记忆
AND 805.09  ; RK_05 #1入壳铝壳有料感应标志[0005.09]
ANDNOT H31.00  ; RK_05 #1入壳机构有电池记忆
ANDNOT H31.04  ; RK_05 #1入壳机构入壳中记忆
LDNOT H31.02  ; RK_05 #1入壳机构有铝壳记忆
LD 805.09  ; RK_05 #1入壳铝壳有料感应标志[0005.09]
AND H31.00  ; RK_05 #1入壳机构有电池记忆
LDNOT 805.09  ; RK_05 #1入壳铝壳有料感应标志[0005.09]
ANDNOT H31.00  ; RK_05 #1入壳机构有电池记忆
ORLD
ANDLD
LDNOT H36.04  ; RK_05 #2入壳机构入壳中记忆
ANDNOT H36.02  ; RK_05 #2入壳机构有铝壳记忆
LD 805.11  ; RK_05 #2入壳铝壳有料感应标志[0005.11]
AND H36.00  ; RK_05 #2入壳机构有电池记忆
LDNOT 805.11  ; RK_05 #2入壳铝壳有料感应标志[0005.11]
ANDNOT H36.00  ; RK_05 #2入壳机构有电池记忆
ORLD
ANDLD
OR H36.04  ; RK_05 #2入壳机构入壳中记忆
OR H7.04  ; #2入壳机构屏蔽
ANDLD
ORLD
ANDLD
ANDNOT H7.03  ; #1入壳机构屏蔽
OUT W214.03  ; 电芯上料X轴去#1入壳放料位条件

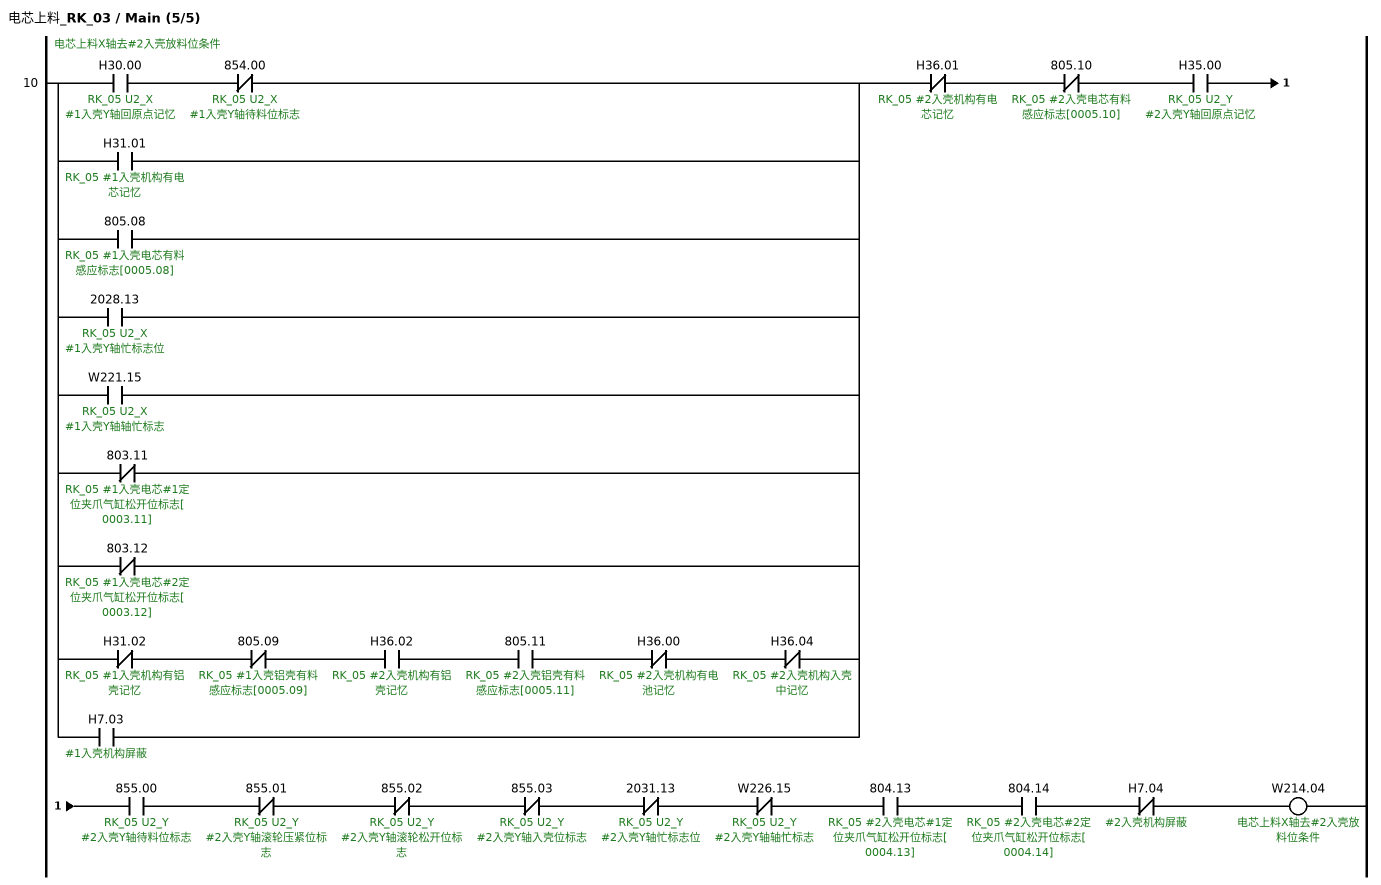
; rung 10: 电芯上料X轴去#2入壳放料位条件
LD H30.00  ; RK_05 U2_X #1入壳Y轴回原点记忆
ANDNOT 854.00  ; RK_05 U2_X #1入壳Y轴待料位标志
OR H31.01  ; RK_05 #1入壳机构有电芯记忆
OR 805.08  ; RK_05 #1入壳电芯有料感应标志[0005.08]
OR 2028.13  ; RK_05 U2_X #1入壳Y轴忙标志位
OR W221.15  ; RK_05 U2_X #1入壳Y轴轴忙标志
ORNOT 803.11  ; RK_05 #1入壳电芯#1定位夹爪气缸松开位标志[0003.11]
ORNOT 803.12  ; RK_05 #1入壳电芯#2定位夹爪气缸松开位标志[0003.12]
LDNOT H31.02  ; RK_05 #1入壳机构有铝壳记忆
ANDNOT 805.09  ; RK_05 #1入壳铝壳有料感应标志[0005.09]
AND H36.02  ; RK_05 #2入壳机构有铝壳记忆
AND 805.11  ; RK_05 #2入壳铝壳有料感应标志[0005.11]
ANDNOT H36.00  ; RK_05 #2入壳机构有电池记忆
ANDNOT H36.04  ; RK_05 #2入壳机构入壳中记忆
ORLD
OR H7.03  ; #1入壳机构屏蔽
ANDNOT H36.01  ; RK_05 #2入壳机构有电芯记忆
ANDNOT 805.10  ; RK_05 #2入壳电芯有料感应标志[0005.10]
AND H35.00  ; RK_05 U2_Y #2入壳Y轴回原点记忆
AND 855.00  ; RK_05 U2_Y #2入壳Y轴待料位标志
ANDNOT 855.01  ; RK_05 U2_Y #2入壳Y轴滚轮压紧位标志
ANDNOT 855.02  ; RK_05 U2_Y #2入壳Y轴滚轮松开位标志
ANDNOT 855.03  ; RK_05 U2_Y #2入壳Y轴入壳位标志
ANDNOT 2031.13  ; RK_05 U2_Y #2入壳Y轴忙标志位
ANDNOT W226.15  ; RK_05 U2_Y #2入壳Y轴轴忙标志
AND 804.13  ; RK_05 #2入壳电芯#1定位夹爪气缸松开位标志[0004.13]
AND 804.14  ; RK_05 #2入壳电芯#2定位夹爪气缸松开位标志[0004.14]
ANDNOT H7.04  ; #2入壳机构屏蔽
OUT W214.04  ; 电芯上料X轴去#2入壳放料位条件

### Section 手动

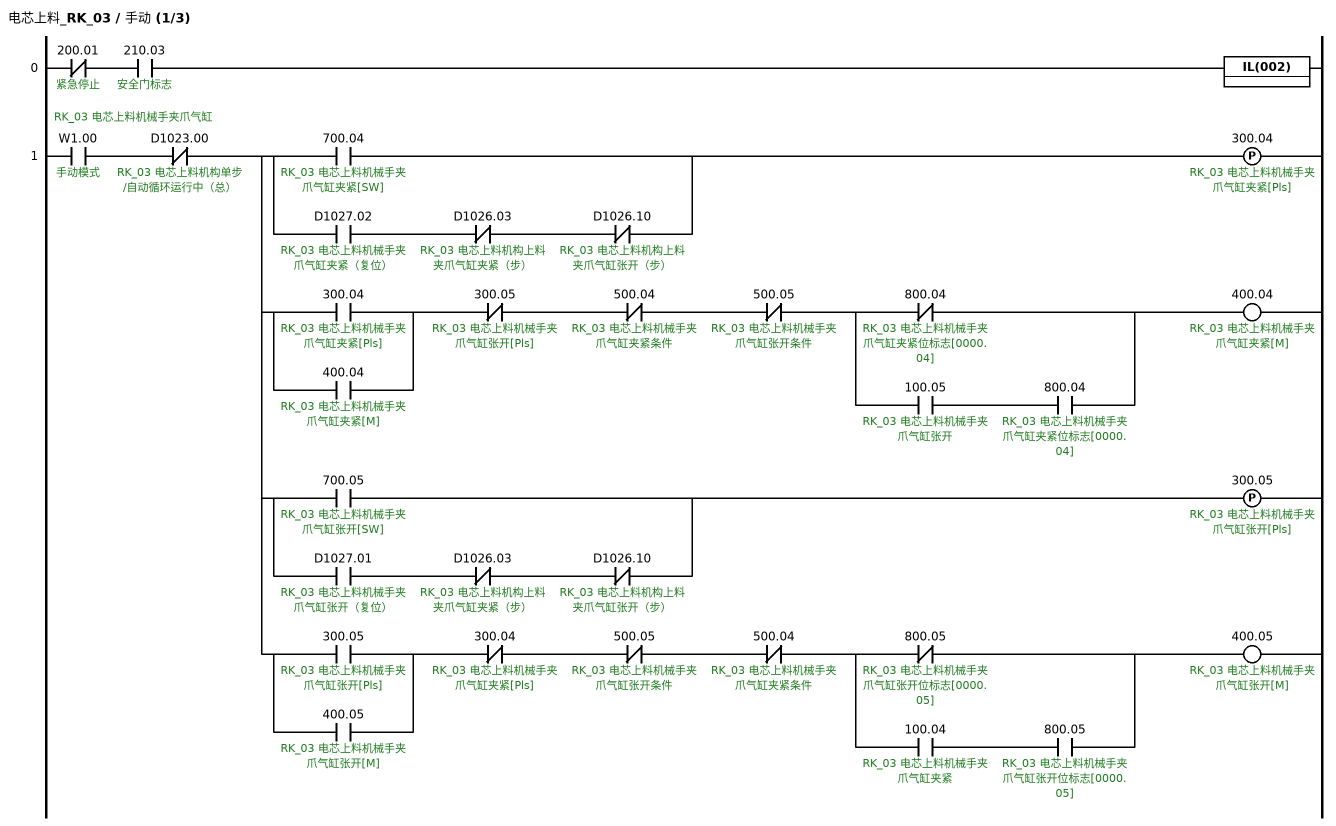
; rung 0
LDNOT 200.01  ; 紧急停止
AND 210.03  ; 安全门标志
IL(002)
; rung 1: RK_03 电芯上料机械手夹爪气缸
LD W1.00  ; 手动模式
ANDNOT D1023.00  ; RK_03 电芯上料机构单步/自动循环运行中（总）
OUT TR0
LD 700.04  ; RK_03 电芯上料机械手夹爪气缸夹紧[SW]
LD D1027.02  ; RK_03 电芯上料机械手夹爪气缸夹紧（复位）
ANDNOT D1026.03  ; RK_03 电芯上料机构上料夹爪气缸夹紧（步）
ANDNOT D1026.10  ; RK_03 电芯上料机构上料夹爪气缸张开（步）
ORLD
ANDLD
DIFU(013) 300.04  ; RK_03 电芯上料机械手夹爪气缸夹紧[Pls]
LD TR0
LD 300.04  ; RK_03 电芯上料机械手夹爪气缸夹紧[Pls]
OR 400.04  ; RK_03 电芯上料机械手夹爪气缸夹紧[M]
ANDLD
ANDNOT 300.05  ; RK_03 电芯上料机械手夹爪气缸张开[Pls]
ANDNOT 500.04  ; RK_03 电芯上料机械手夹爪气缸夹紧条件
ANDNOT 500.05  ; RK_03 电芯上料机械手夹爪气缸张开条件
LDNOT 800.04  ; RK_03 电芯上料机械手夹爪气缸夹紧位标志[0000.04]
LD 100.05  ; RK_03 电芯上料机械手夹爪气缸张开
AND 800.04  ; RK_03 电芯上料机械手夹爪气缸夹紧位标志[0000.04]
ORLD
ANDLD
OUT 400.04  ; RK_03 电芯上料机械手夹爪气缸夹紧[M]
LD TR0
LD 700.05  ; RK_03 电芯上料机械手夹爪气缸张开[SW]
LD D1027.01  ; RK_03 电芯上料机械手夹爪气缸张开（复位）
ANDNOT D1026.03  ; RK_03 电芯上料机构上料夹爪气缸夹紧（步）
ANDNOT D1026.10  ; RK_03 电芯上料机构上料夹爪气缸张开（步）
ORLD
ANDLD
DIFU(013) 300.05  ; RK_03 电芯上料机械手夹爪气缸张开[Pls]
LD TR0
LD 300.05  ; RK_03 电芯上料机械手夹爪气缸张开[Pls]
OR 400.05  ; RK_03 电芯上料机械手夹爪气缸张开[M]
ANDLD
ANDNOT 300.04  ; RK_03 电芯上料机械手夹爪气缸夹紧[Pls]
ANDNOT 500.05  ; RK_03 电芯上料机械手夹爪气缸张开条件
ANDNOT 500.04  ; RK_03 电芯上料机械手夹爪气缸夹紧条件
LDNOT 800.05  ; RK_03 电芯上料机械手夹爪气缸张开位标志[0000.05]
LD 100.04  ; RK_03 电芯上料机械手夹爪气缸夹紧
AND 800.05  ; RK_03 电芯上料机械手夹爪气缸张开位标志[0000.05]
ORLD
ANDLD
OUT 400.05  ; RK_03 电芯上料机械手夹爪气缸张开[M]

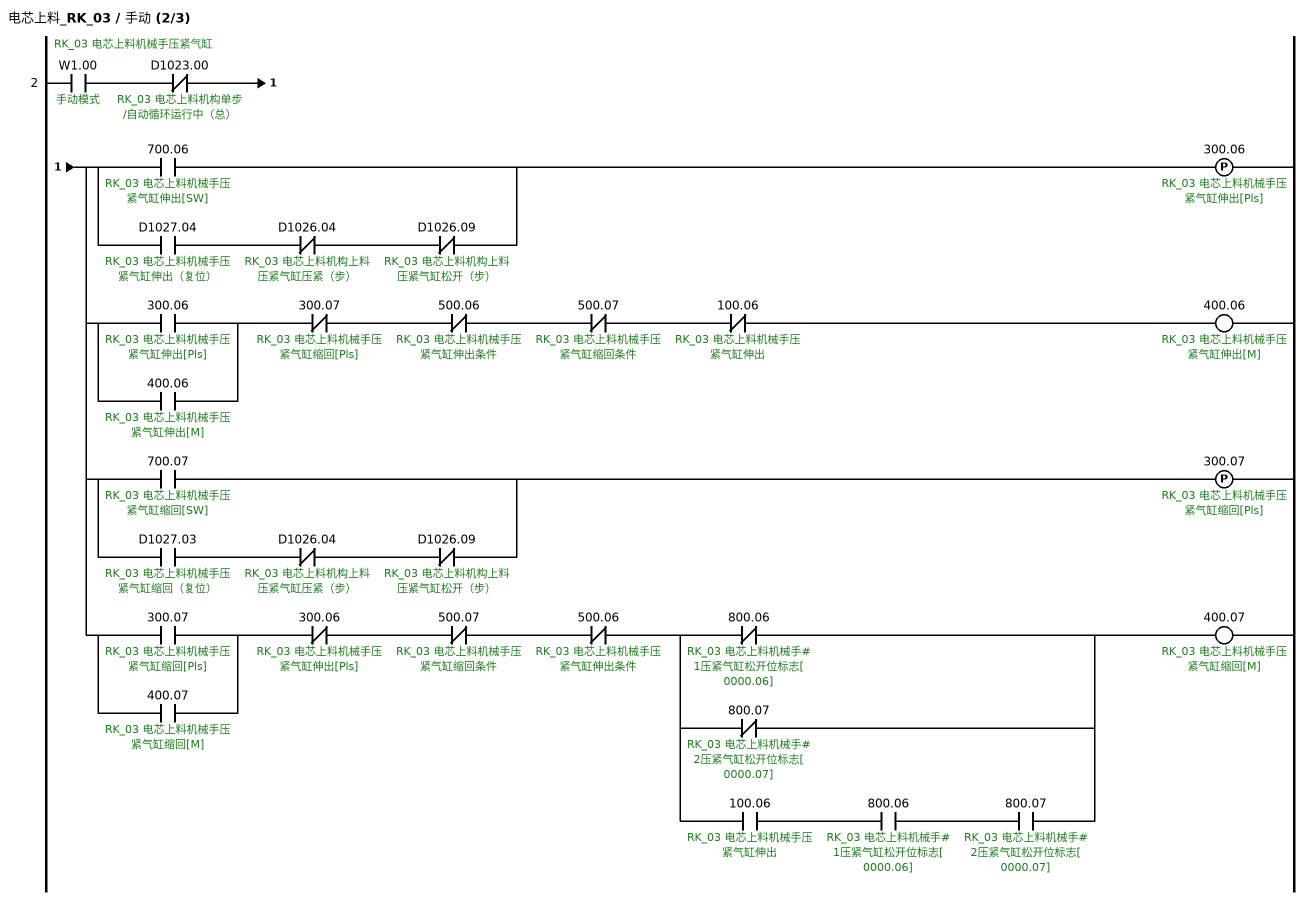
; rung 2: RK_03 电芯上料机械手压紧气缸
LD W1.00  ; 手动模式
ANDNOT D1023.00  ; RK_03 电芯上料机构单步/自动循环运行中（总）
OUT TR0
LD 700.06  ; RK_03 电芯上料机械手压紧气缸伸出[SW]
LD D1027.04  ; RK_03 电芯上料机械手压紧气缸伸出（复位）
ANDNOT D1026.04  ; RK_03 电芯上料机构上料压紧气缸压紧（步）
ANDNOT D1026.09  ; RK_03 电芯上料机构上料压紧气缸松开（步）
ORLD
ANDLD
DIFU(013) 300.06  ; RK_03 电芯上料机械手压紧气缸伸出[Pls]
LD TR0
LD 300.06  ; RK_03 电芯上料机械手压紧气缸伸出[Pls]
OR 400.06  ; RK_03 电芯上料机械手压紧气缸伸出[M]
ANDLD
ANDNOT 300.07  ; RK_03 电芯上料机械手压紧气缸缩回[Pls]
ANDNOT 500.06  ; RK_03 电芯上料机械手压紧气缸伸出条件
ANDNOT 500.07  ; RK_03 电芯上料机械手压紧气缸缩回条件
ANDNOT 100.06  ; RK_03 电芯上料机械手压紧气缸伸出
OUT 400.06  ; RK_03 电芯上料机械手压紧气缸伸出[M]
LD TR0
LD 700.07  ; RK_03 电芯上料机械手压紧气缸缩回[SW]
LD D1027.03  ; RK_03 电芯上料机械手压紧气缸缩回（复位）
ANDNOT D1026.04  ; RK_03 电芯上料机构上料压紧气缸压紧（步）
ANDNOT D1026.09  ; RK_03 电芯上料机构上料压紧气缸松开（步）
ORLD
ANDLD
DIFU(013) 300.07  ; RK_03 电芯上料机械手压紧气缸缩回[Pls]
LD TR0
LD 300.07  ; RK_03 电芯上料机械手压紧气缸缩回[Pls]
OR 400.07  ; RK_03 电芯上料机械手压紧气缸缩回[M]
ANDLD
ANDNOT 300.06  ; RK_03 电芯上料机械手压紧气缸伸出[Pls]
ANDNOT 500.07  ; RK_03 电芯上料机械手压紧气缸缩回条件
ANDNOT 500.06  ; RK_03 电芯上料机械手压紧气缸伸出条件
LDNOT 800.06  ; RK_03 电芯上料机械手#1压紧气缸松开位标志[0000.06]
ORNOT 800.07  ; RK_03 电芯上料机械手#2压紧气缸松开位标志[0000.07]
LD 100.06  ; RK_03 电芯上料机械手压紧气缸伸出
AND 800.06  ; RK_03 电芯上料机械手#1压紧气缸松开位标志[0000.06]
AND 800.07  ; RK_03 电芯上料机械手#2压紧气缸松开位标志[0000.07]
ORLD
ANDLD
OUT 400.07  ; RK_03 电芯上料机械手压紧气缸缩回[M]

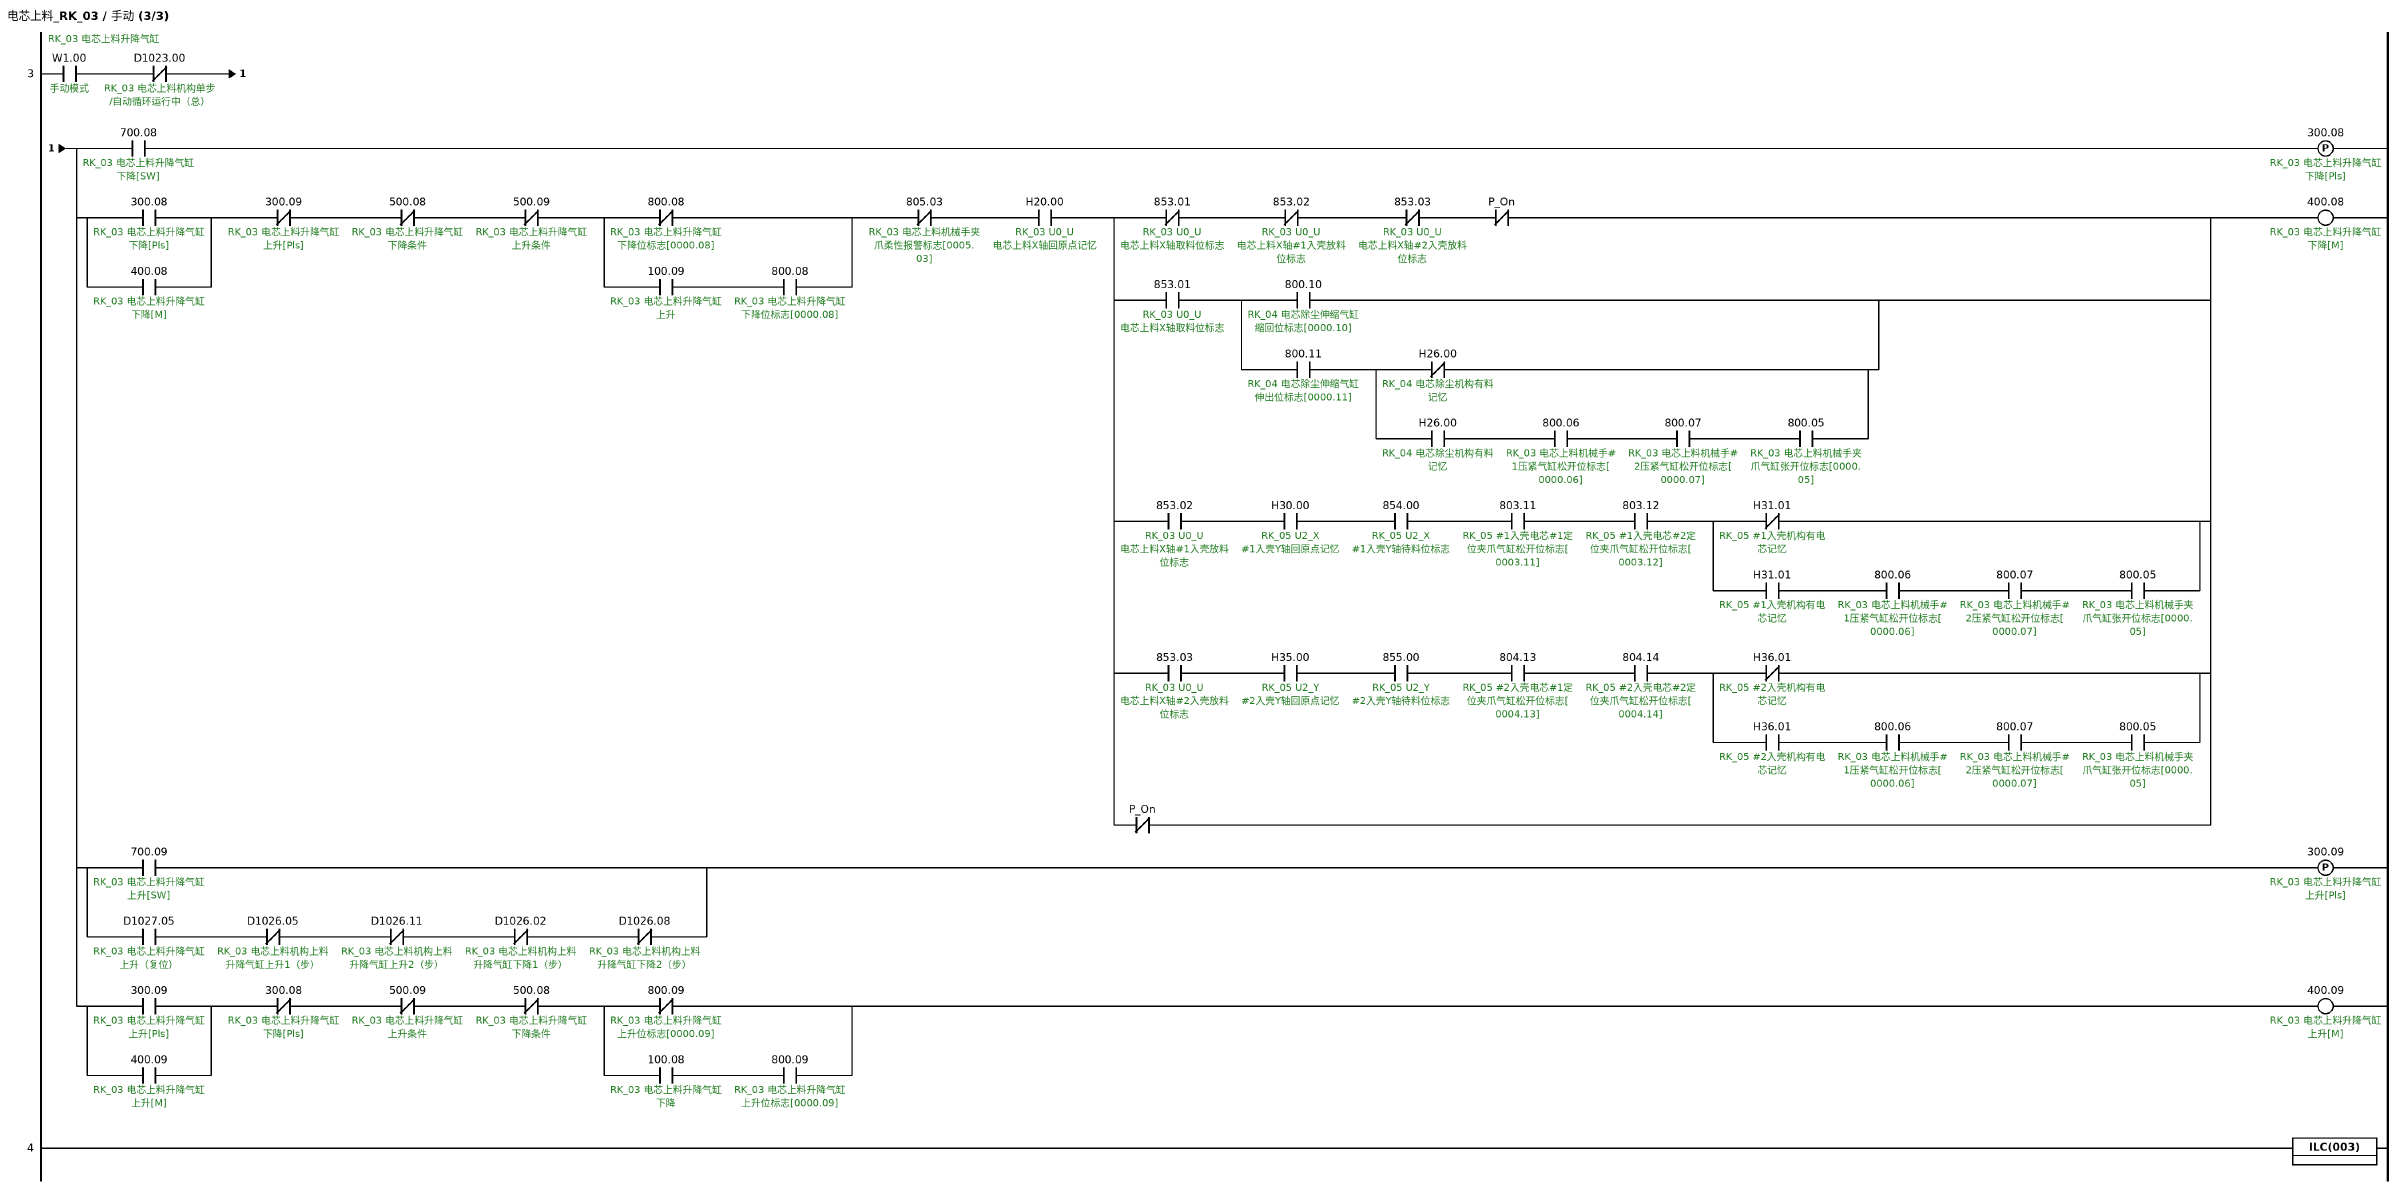
; rung 3: RK_03 电芯上料升降气缸
LD W1.00  ; 手动模式
ANDNOT D1023.00  ; RK_03 电芯上料机构单步/自动循环运行中（总）
OUT TR0
AND 700.08  ; RK_03 电芯上料升降气缸下降[SW]
DIFU(013) 300.08  ; RK_03 电芯上料升降气缸下降[Pls]
LD TR0
LD 300.08  ; RK_03 电芯上料升降气缸下降[Pls]
OR 400.08  ; RK_03 电芯上料升降气缸下降[M]
ANDLD
ANDNOT 300.09  ; RK_03 电芯上料升降气缸上升[Pls]
ANDNOT 500.08  ; RK_03 电芯上料升降气缸下降条件
ANDNOT 500.09  ; RK_03 电芯上料升降气缸上升条件
LDNOT 800.08  ; RK_03 电芯上料升降气缸下降位标志[0000.08]
LD 100.09  ; RK_03 电芯上料升降气缸上升
AND 800.08  ; RK_03 电芯上料升降气缸下降位标志[0000.08]
ORLD
ANDLD
ANDNOT 805.03  ; RK_03 电芯上料机械手夹爪柔性报警标志[0005.03]
AND H20.00  ; RK_03 U0_U 电芯上料X轴回原点记忆
LDNOT 853.01  ; RK_03 U0_U 电芯上料X轴取料位标志
ANDNOT 853.02  ; RK_03 U0_U 电芯上料X轴#1入壳放料位标志
ANDNOT 853.03  ; RK_03 U0_U 电芯上料X轴#2入壳放料位标志
ANDNOT P_On
LD 853.01  ; RK_03 U0_U 电芯上料X轴取料位标志
LD 800.10  ; RK_04 电芯除尘伸缩气缸缩回位标志[0000.10]
LD 800.11  ; RK_04 电芯除尘伸缩气缸伸出位标志[0000.11]
LDNOT H26.00  ; RK_04 电芯除尘机构有料记忆
LD H26.00  ; RK_04 电芯除尘机构有料记忆
AND 800.06  ; RK_03 电芯上料机械手#1压紧气缸松开位标志[0000.06]
AND 800.07  ; RK_03 电芯上料机械手#2压紧气缸松开位标志[0000.07]
AND 800.05  ; RK_03 电芯上料机械手夹爪气缸张开位标志[0000.05]
ORLD
ANDLD
ORLD
ANDLD
ORLD
LD 853.02  ; RK_03 U0_U 电芯上料X轴#1入壳放料位标志
AND H30.00  ; RK_05 U2_X #1入壳Y轴回原点记忆
AND 854.00  ; RK_05 U2_X #1入壳Y轴待料位标志
AND 803.11  ; RK_05 #1入壳电芯#1定位夹爪气缸松开位标志[0003.11]
AND 803.12  ; RK_05 #1入壳电芯#2定位夹爪气缸松开位标志[0003.12]
LDNOT H31.01  ; RK_05 #1入壳机构有电芯记忆
LD H31.01  ; RK_05 #1入壳机构有电芯记忆
AND 800.06  ; RK_03 电芯上料机械手#1压紧气缸松开位标志[0000.06]
AND 800.07  ; RK_03 电芯上料机械手#2压紧气缸松开位标志[0000.07]
AND 800.05  ; RK_03 电芯上料机械手夹爪气缸张开位标志[0000.05]
ORLD
ANDLD
ORLD
LD 853.03  ; RK_03 U0_U 电芯上料X轴#2入壳放料位标志
AND H35.00  ; RK_05 U2_Y #2入壳Y轴回原点记忆
AND 855.00  ; RK_05 U2_Y #2入壳Y轴待料位标志
AND 804.13  ; RK_05 #2入壳电芯#1定位夹爪气缸松开位标志[0004.13]
AND 804.14  ; RK_05 #2入壳电芯#2定位夹爪气缸松开位标志[0004.14]
LDNOT H36.01  ; RK_05 #2入壳机构有电芯记忆
LD H36.01  ; RK_05 #2入壳机构有电芯记忆
AND 800.06  ; RK_03 电芯上料机械手#1压紧气缸松开位标志[0000.06]
AND 800.07  ; RK_03 电芯上料机械手#2压紧气缸松开位标志[0000.07]
AND 800.05  ; RK_03 电芯上料机械手夹爪气缸张开位标志[0000.05]
ORLD
ANDLD
ORLD
ORNOT P_On
ANDLD
OUT 400.08  ; RK_03 电芯上料升降气缸下降[M]
LD TR0
LD 700.09  ; RK_03 电芯上料升降气缸上升[SW]
LD D1027.05  ; RK_03 电芯上料升降气缸上升（复位）
ANDNOT D1026.05  ; RK_03 电芯上料机构上料升降气缸上升1（步）
ANDNOT D1026.11  ; RK_03 电芯上料机构上料升降气缸上升2（步）
ANDNOT D1026.02  ; RK_03 电芯上料机构上料升降气缸下降1（步）
ANDNOT D1026.08  ; RK_03 电芯上料机构上料升降气缸下降2（步）
ORLD
ANDLD
DIFU(013) 300.09  ; RK_03 电芯上料升降气缸上升[Pls]
LD TR0
LD 300.09  ; RK_03 电芯上料升降气缸上升[Pls]
OR 400.09  ; RK_03 电芯上料升降气缸上升[M]
ANDLD
ANDNOT 300.08  ; RK_03 电芯上料升降气缸下降[Pls]
ANDNOT 500.09  ; RK_03 电芯上料升降气缸上升条件
ANDNOT 500.08  ; RK_03 电芯上料升降气缸下降条件
LDNOT 800.09  ; RK_03 电芯上料升降气缸上升位标志[0000.09]
LD 100.08  ; RK_03 电芯上料升降气缸下降
AND 800.09  ; RK_03 电芯上料升降气缸上升位标志[0000.09]
ORLD
ANDLD
OUT 400.09  ; RK_03 电芯上料升降气缸上升[M]
; rung 4
ILC(003)

### Section 自动

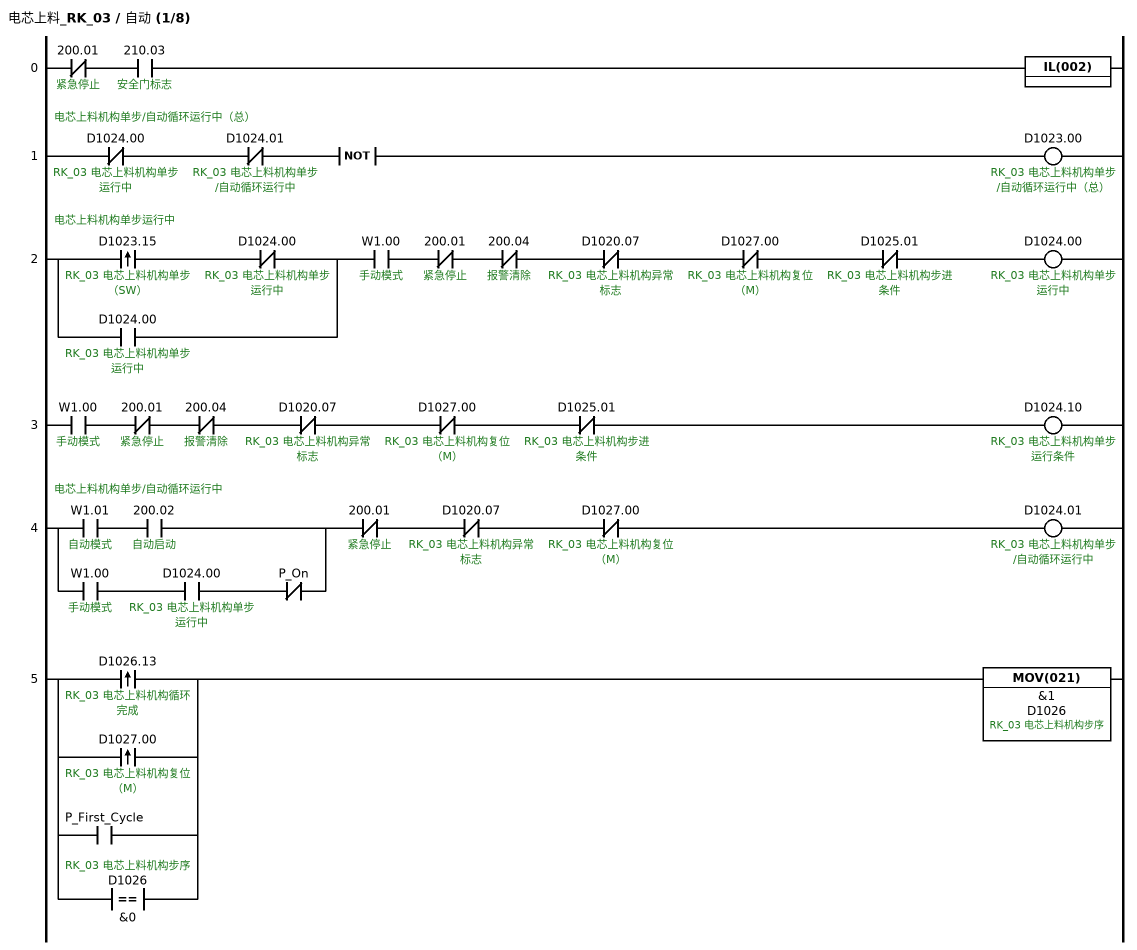
; rung 0
LDNOT 200.01  ; 紧急停止
AND 210.03  ; 安全门标志
IL(002)
; rung 1: 电芯上料机构单步/自动循环运行中（总）
LDNOT D1024.00  ; RK_03 电芯上料机构单步运行中
ANDNOT D1024.01  ; RK_03 电芯上料机构单步/自动循环运行中
NOT(520)
OUT D1023.00  ; RK_03 电芯上料机构单步/自动循环运行中（总）
; rung 2: 电芯上料机构单步运行中
@LD D1023.15  ; RK_03 电芯上料机构单步（SW）
ANDNOT D1024.00  ; RK_03 电芯上料机构单步运行中
OR D1024.00  ; RK_03 电芯上料机构单步运行中
AND W1.00  ; 手动模式
ANDNOT 200.01  ; 紧急停止
ANDNOT 200.04  ; 报警清除
ANDNOT D1020.07  ; RK_03 电芯上料机构异常标志
ANDNOT D1027.00  ; RK_03 电芯上料机构复位（M）
ANDNOT D1025.01  ; RK_03 电芯上料机构步进条件
OUT D1024.00  ; RK_03 电芯上料机构单步运行中
; rung 3
LD W1.00  ; 手动模式
ANDNOT 200.01  ; 紧急停止
ANDNOT 200.04  ; 报警清除
ANDNOT D1020.07  ; RK_03 电芯上料机构异常标志
ANDNOT D1027.00  ; RK_03 电芯上料机构复位（M）
ANDNOT D1025.01  ; RK_03 电芯上料机构步进条件
OUT D1024.10  ; RK_03 电芯上料机构单步运行条件
; rung 4: 电芯上料机构单步/自动循环运行中
LD W1.01  ; 自动模式
AND 200.02  ; 自动启动
LD W1.00  ; 手动模式
AND D1024.00  ; RK_03 电芯上料机构单步运行中
ANDNOT P_On
ORLD
ANDNOT 200.01  ; 紧急停止
ANDNOT D1020.07  ; RK_03 电芯上料机构异常标志
ANDNOT D1027.00  ; RK_03 电芯上料机构复位（M）
OUT D1024.01  ; RK_03 电芯上料机构单步/自动循环运行中
; rung 5
@LD D1026.13  ; RK_03 电芯上料机构循环完成
@OR D1027.00  ; RK_03 电芯上料机构复位（M）
OR P_First_Cycle
OR=(300) D1026 &0  ; RK_03 电芯上料机构步序
MOV(021) &1 D1026  ; RK_03 电芯上料机构步序

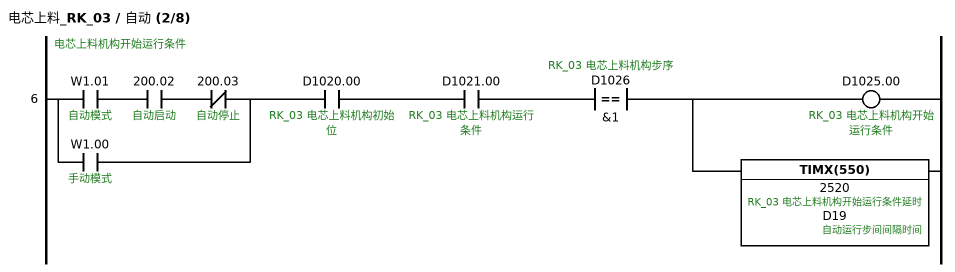
; rung 6: 电芯上料机构开始运行条件
LD W1.01  ; 自动模式
AND 200.02  ; 自动启动
ANDNOT 200.03  ; 自动停止
OR W1.00  ; 手动模式
AND D1020.00  ; RK_03 电芯上料机构初始位
AND D1021.00  ; RK_03 电芯上料机构运行条件
AND=(300) D1026 &1  ; RK_03 电芯上料机构步序
OUT D1025.00  ; RK_03 电芯上料机构开始运行条件
TIMX(550) 2520 D19  ; 自动运行步间间隔时间, RK_03 电芯上料机构开始运行条件延时

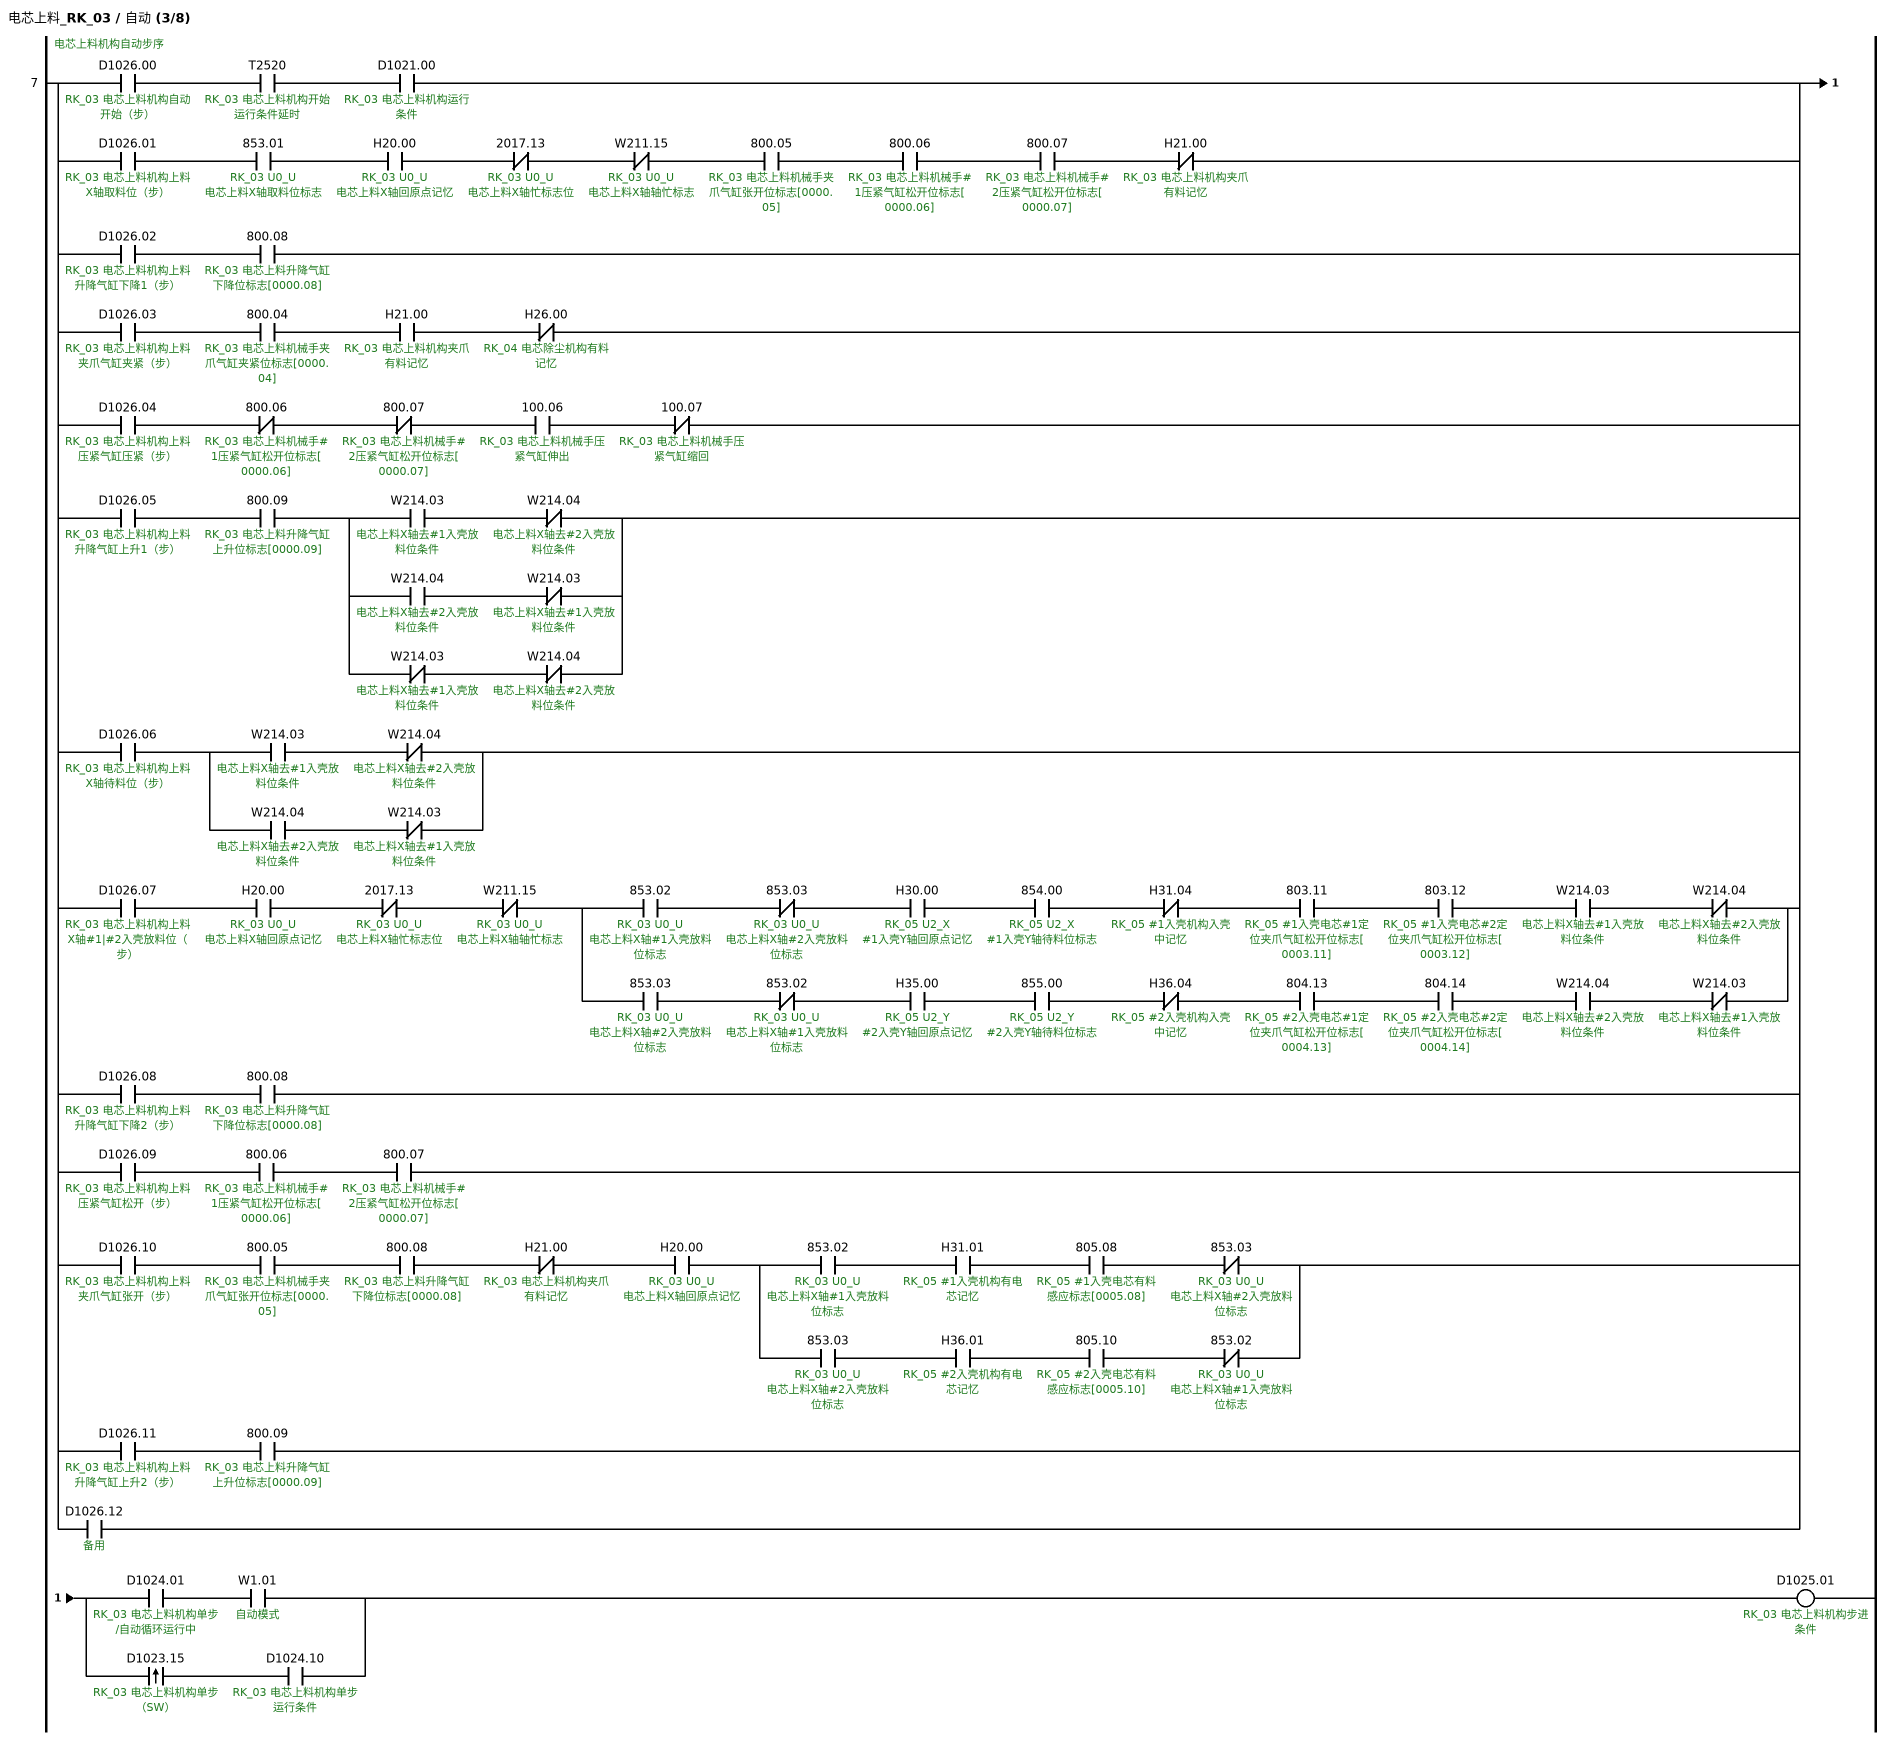
; rung 7: 电芯上料机构自动步序
LD D1026.00  ; RK_03 电芯上料机构自动开始（步）
AND T2520  ; RK_03 电芯上料机构开始运行条件延时
AND D1021.00  ; RK_03 电芯上料机构运行条件
LD D1026.01  ; RK_03 电芯上料机构上料X轴取料位（步）
AND 853.01  ; RK_03 U0_U 电芯上料X轴取料位标志
AND H20.00  ; RK_03 U0_U 电芯上料X轴回原点记忆
ANDNOT 2017.13  ; RK_03 U0_U 电芯上料X轴忙标志位
ANDNOT W211.15  ; RK_03 U0_U 电芯上料X轴轴忙标志
AND 800.05  ; RK_03 电芯上料机械手夹爪气缸张开位标志[0000.05]
AND 800.06  ; RK_03 电芯上料机械手#1压紧气缸松开位标志[0000.06]
AND 800.07  ; RK_03 电芯上料机械手#2压紧气缸松开位标志[0000.07]
ANDNOT H21.00  ; RK_03 电芯上料机构夹爪有料记忆
ORLD
LD D1026.02  ; RK_03 电芯上料机构上料升降气缸下降1（步）
AND 800.08  ; RK_03 电芯上料升降气缸下降位标志[0000.08]
ORLD
LD D1026.03  ; RK_03 电芯上料机构上料夹爪气缸夹紧（步）
AND 800.04  ; RK_03 电芯上料机械手夹爪气缸夹紧位标志[0000.04]
AND H21.00  ; RK_03 电芯上料机构夹爪有料记忆
ANDNOT H26.00  ; RK_04 电芯除尘机构有料记忆
ORLD
LD D1026.04  ; RK_03 电芯上料机构上料压紧气缸压紧（步）
ANDNOT 800.06  ; RK_03 电芯上料机械手#1压紧气缸松开位标志[0000.06]
ANDNOT 800.07  ; RK_03 电芯上料机械手#2压紧气缸松开位标志[0000.07]
AND 100.06  ; RK_03 电芯上料机械手压紧气缸伸出
ANDNOT 100.07  ; RK_03 电芯上料机械手压紧气缸缩回
ORLD
LD D1026.05  ; RK_03 电芯上料机构上料升降气缸上升1（步）
AND 800.09  ; RK_03 电芯上料升降气缸上升位标志[0000.09]
LD W214.03  ; 电芯上料X轴去#1入壳放料位条件
ANDNOT W214.04  ; 电芯上料X轴去#2入壳放料位条件
LD W214.04  ; 电芯上料X轴去#2入壳放料位条件
ANDNOT W214.03  ; 电芯上料X轴去#1入壳放料位条件
ORLD
LDNOT W214.03  ; 电芯上料X轴去#1入壳放料位条件
ANDNOT W214.04  ; 电芯上料X轴去#2入壳放料位条件
ORLD
ANDLD
ORLD
LD D1026.06  ; RK_03 电芯上料机构上料X轴待料位（步）
LD W214.03  ; 电芯上料X轴去#1入壳放料位条件
ANDNOT W214.04  ; 电芯上料X轴去#2入壳放料位条件
LD W214.04  ; 电芯上料X轴去#2入壳放料位条件
ANDNOT W214.03  ; 电芯上料X轴去#1入壳放料位条件
ORLD
ANDLD
ORLD
LD D1026.07  ; RK_03 电芯上料机构上料X轴#1|#2入壳放料位（步）
AND H20.00  ; RK_03 U0_U 电芯上料X轴回原点记忆
ANDNOT 2017.13  ; RK_03 U0_U 电芯上料X轴忙标志位
ANDNOT W211.15  ; RK_03 U0_U 电芯上料X轴轴忙标志
LD 853.02  ; RK_03 U0_U 电芯上料X轴#1入壳放料位标志
ANDNOT 853.03  ; RK_03 U0_U 电芯上料X轴#2入壳放料位标志
AND H30.00  ; RK_05 U2_X #1入壳Y轴回原点记忆
AND 854.00  ; RK_05 U2_X #1入壳Y轴待料位标志
ANDNOT H31.04  ; RK_05 #1入壳机构入壳中记忆
AND 803.11  ; RK_05 #1入壳电芯#1定位夹爪气缸松开位标志[0003.11]
AND 803.12  ; RK_05 #1入壳电芯#2定位夹爪气缸松开位标志[0003.12]
AND W214.03  ; 电芯上料X轴去#1入壳放料位条件
ANDNOT W214.04  ; 电芯上料X轴去#2入壳放料位条件
LD 853.03  ; RK_03 U0_U 电芯上料X轴#2入壳放料位标志
ANDNOT 853.02  ; RK_03 U0_U 电芯上料X轴#1入壳放料位标志
AND H35.00  ; RK_05 U2_Y #2入壳Y轴回原点记忆
AND 855.00  ; RK_05 U2_Y #2入壳Y轴待料位标志
ANDNOT H36.04  ; RK_05 #2入壳机构入壳中记忆
AND 804.13  ; RK_05 #2入壳电芯#1定位夹爪气缸松开位标志[0004.13]
AND 804.14  ; RK_05 #2入壳电芯#2定位夹爪气缸松开位标志[0004.14]
AND W214.04  ; 电芯上料X轴去#2入壳放料位条件
ANDNOT W214.03  ; 电芯上料X轴去#1入壳放料位条件
ORLD
ANDLD
ORLD
LD D1026.08  ; RK_03 电芯上料机构上料升降气缸下降2（步）
AND 800.08  ; RK_03 电芯上料升降气缸下降位标志[0000.08]
ORLD
LD D1026.09  ; RK_03 电芯上料机构上料压紧气缸松开（步）
AND 800.06  ; RK_03 电芯上料机械手#1压紧气缸松开位标志[0000.06]
AND 800.07  ; RK_03 电芯上料机械手#2压紧气缸松开位标志[0000.07]
ORLD
LD D1026.10  ; RK_03 电芯上料机构上料夹爪气缸张开（步）
AND 800.05  ; RK_03 电芯上料机械手夹爪气缸张开位标志[0000.05]
AND 800.08  ; RK_03 电芯上料升降气缸下降位标志[0000.08]
ANDNOT H21.00  ; RK_03 电芯上料机构夹爪有料记忆
AND H20.00  ; RK_03 U0_U 电芯上料X轴回原点记忆
LD 853.02  ; RK_03 U0_U 电芯上料X轴#1入壳放料位标志
AND H31.01  ; RK_05 #1入壳机构有电芯记忆
AND 805.08  ; RK_05 #1入壳电芯有料感应标志[0005.08]
ANDNOT 853.03  ; RK_03 U0_U 电芯上料X轴#2入壳放料位标志
LD 853.03  ; RK_03 U0_U 电芯上料X轴#2入壳放料位标志
AND H36.01  ; RK_05 #2入壳机构有电芯记忆
AND 805.10  ; RK_05 #2入壳电芯有料感应标志[0005.10]
ANDNOT 853.02  ; RK_03 U0_U 电芯上料X轴#1入壳放料位标志
ORLD
ANDLD
ORLD
LD D1026.11  ; RK_03 电芯上料机构上料升降气缸上升2（步）
AND 800.09  ; RK_03 电芯上料升降气缸上升位标志[0000.09]
ORLD
OR D1026.12  ; 备用
LD D1024.01  ; RK_03 电芯上料机构单步/自动循环运行中
AND W1.01  ; 自动模式
@LD D1023.15  ; RK_03 电芯上料机构单步（SW）
AND D1024.10  ; RK_03 电芯上料机构单步运行条件
ORLD
ANDLD
OUT D1025.01  ; RK_03 电芯上料机构步进条件

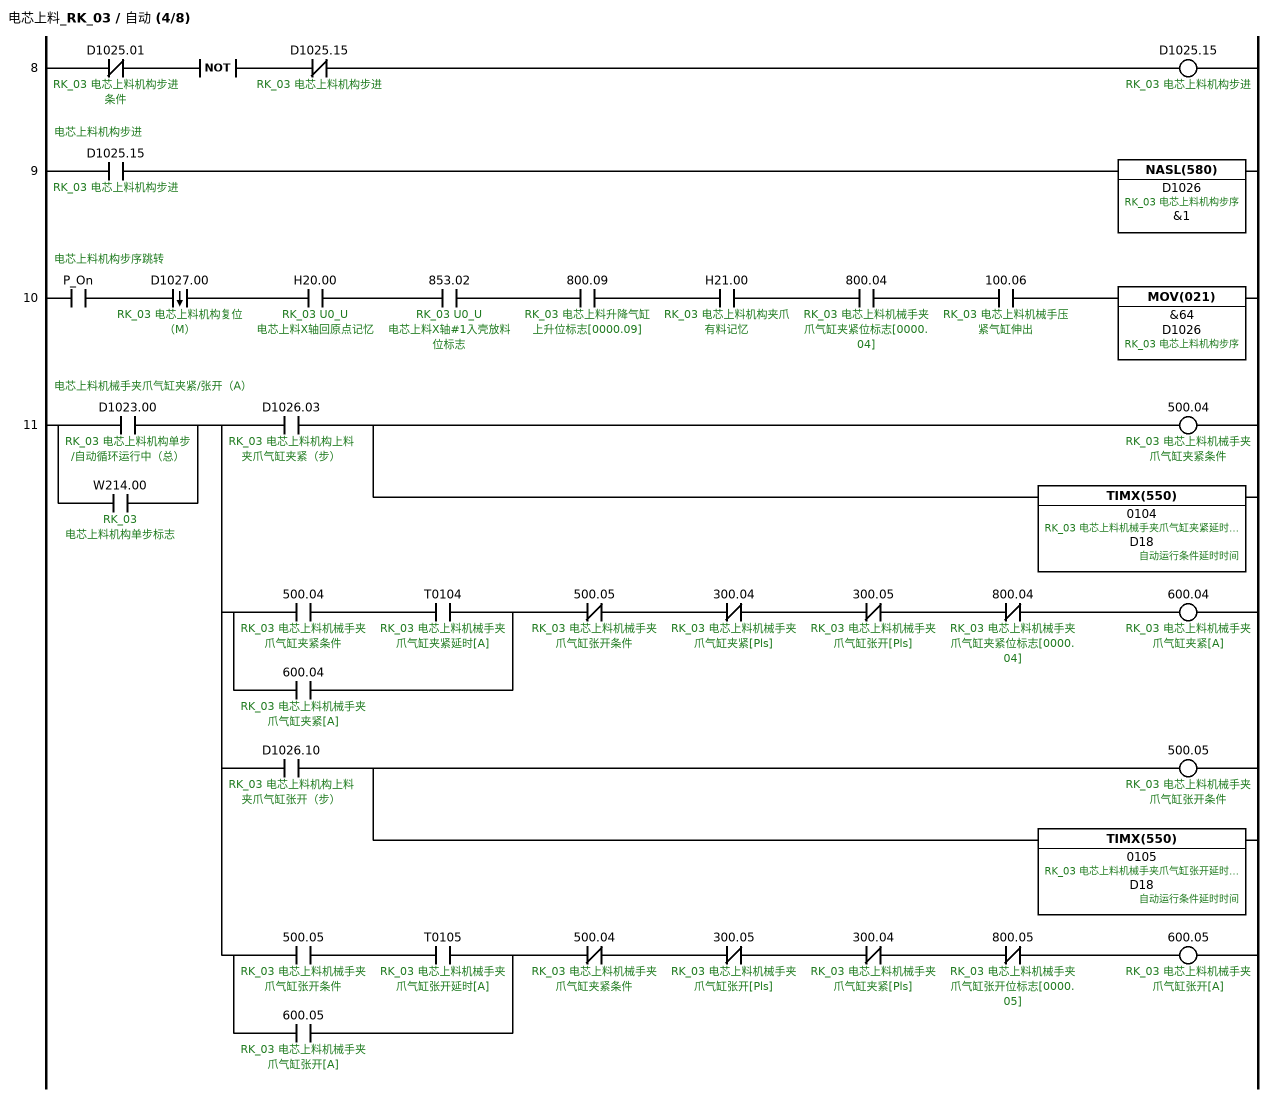
; rung 8
LDNOT D1025.01  ; RK_03 电芯上料机构步进条件
NOT(520)
ANDNOT D1025.15  ; RK_03 电芯上料机构步进
OUT D1025.15  ; RK_03 电芯上料机构步进
; rung 9: 电芯上料机构步进
LD D1025.15  ; RK_03 电芯上料机构步进
NASL(580) D1026 &1  ; RK_03 电芯上料机构步序
; rung 10: 电芯上料机构步序跳转
LD P_On
%AND D1027.00  ; RK_03 电芯上料机构复位（M）
AND H20.00  ; RK_03 U0_U 电芯上料X轴回原点记忆
AND 853.02  ; RK_03 U0_U 电芯上料X轴#1入壳放料位标志
AND 800.09  ; RK_03 电芯上料升降气缸上升位标志[0000.09]
AND H21.00  ; RK_03 电芯上料机构夹爪有料记忆
AND 800.04  ; RK_03 电芯上料机械手夹爪气缸夹紧位标志[0000.04]
AND 100.06  ; RK_03 电芯上料机械手压紧气缸伸出
MOV(021) &64 D1026  ; RK_03 电芯上料机构步序  // RK_03 电芯上料机构上料X轴待料位步（D1026.06）
; rung 11: 电芯上料机械手夹爪气缸夹紧/张开（A）
LD D1023.00  ; RK_03 电芯上料机构单步/自动循环运行中（总）
OR W214.00  ; RK_03  电芯上料机构单步标志
OUT TR0
AND D1026.03  ; RK_03 电芯上料机构上料夹爪气缸夹紧（步）
OUT 500.04  ; RK_03 电芯上料机械手夹爪气缸夹紧条件
TIMX(550) 0104 D18  ; 自动运行条件延时时间, RK_03 电芯上料机械手夹爪气缸夹紧延时[A]
LD TR0
LD 500.04  ; RK_03 电芯上料机械手夹爪气缸夹紧条件
AND T0104  ; RK_03 电芯上料机械手夹爪气缸夹紧延时[A]
OR 600.04  ; RK_03 电芯上料机械手夹爪气缸夹紧[A]
ANDLD
ANDNOT 500.05  ; RK_03 电芯上料机械手夹爪气缸张开条件
ANDNOT 300.04  ; RK_03 电芯上料机械手夹爪气缸夹紧[Pls]
ANDNOT 300.05  ; RK_03 电芯上料机械手夹爪气缸张开[Pls]
ANDNOT 800.04  ; RK_03 电芯上料机械手夹爪气缸夹紧位标志[0000.04]
OUT 600.04  ; RK_03 电芯上料机械手夹爪气缸夹紧[A]
LD TR0
AND D1026.10  ; RK_03 电芯上料机构上料夹爪气缸张开（步）
OUT 500.05  ; RK_03 电芯上料机械手夹爪气缸张开条件
TIMX(550) 0105 D18  ; 自动运行条件延时时间, RK_03 电芯上料机械手夹爪气缸张开延时[A]
LD TR0
LD 500.05  ; RK_03 电芯上料机械手夹爪气缸张开条件
AND T0105  ; RK_03 电芯上料机械手夹爪气缸张开延时[A]
OR 600.05  ; RK_03 电芯上料机械手夹爪气缸张开[A]
ANDLD
ANDNOT 500.04  ; RK_03 电芯上料机械手夹爪气缸夹紧条件
ANDNOT 300.05  ; RK_03 电芯上料机械手夹爪气缸张开[Pls]
ANDNOT 300.04  ; RK_03 电芯上料机械手夹爪气缸夹紧[Pls]
ANDNOT 800.05  ; RK_03 电芯上料机械手夹爪气缸张开位标志[0000.05]
OUT 600.05  ; RK_03 电芯上料机械手夹爪气缸张开[A]

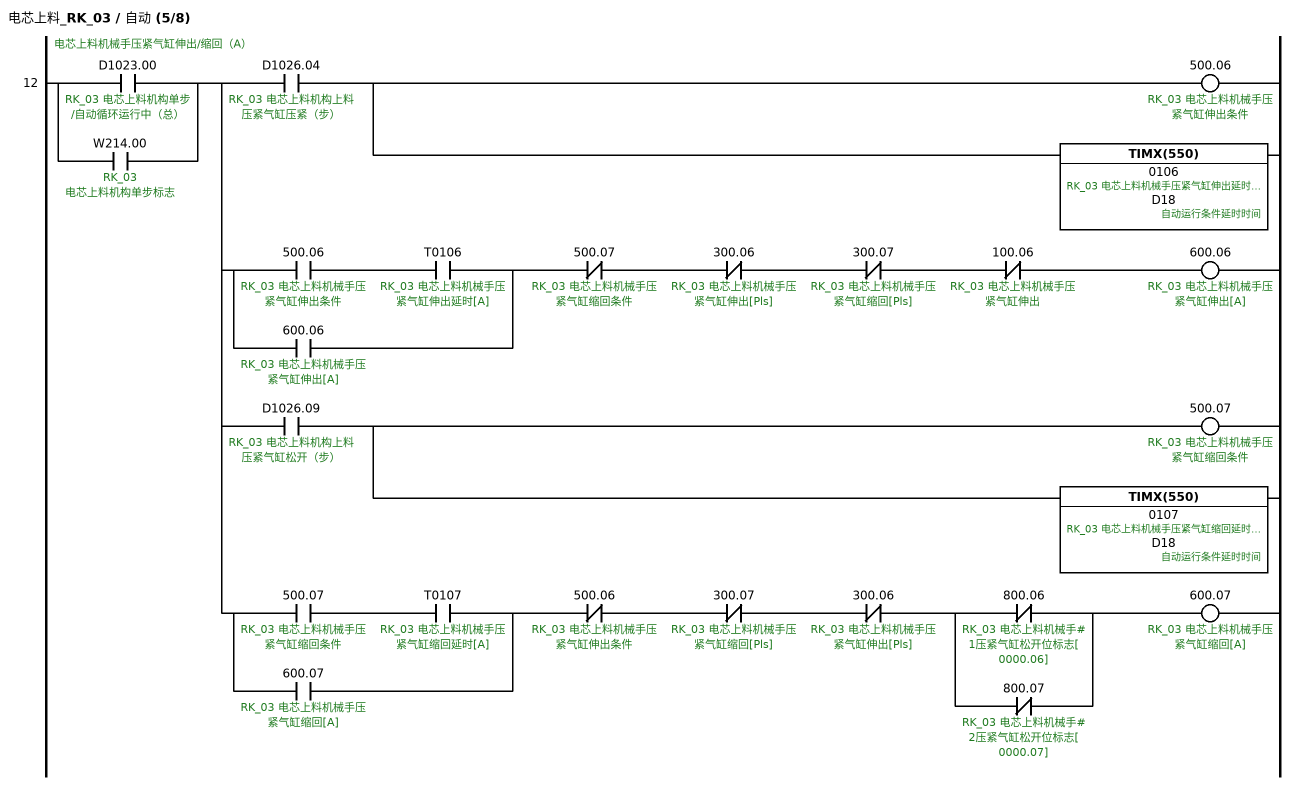
; rung 12: 电芯上料机械手压紧气缸伸出/缩回（A）
LD D1023.00  ; RK_03 电芯上料机构单步/自动循环运行中（总）
OR W214.00  ; RK_03  电芯上料机构单步标志
OUT TR0
AND D1026.04  ; RK_03 电芯上料机构上料压紧气缸压紧（步）
OUT 500.06  ; RK_03 电芯上料机械手压紧气缸伸出条件
TIMX(550) 0106 D18  ; 自动运行条件延时时间, RK_03 电芯上料机械手压紧气缸伸出延时[A]
LD TR0
LD 500.06  ; RK_03 电芯上料机械手压紧气缸伸出条件
AND T0106  ; RK_03 电芯上料机械手压紧气缸伸出延时[A]
OR 600.06  ; RK_03 电芯上料机械手压紧气缸伸出[A]
ANDLD
ANDNOT 500.07  ; RK_03 电芯上料机械手压紧气缸缩回条件
ANDNOT 300.06  ; RK_03 电芯上料机械手压紧气缸伸出[Pls]
ANDNOT 300.07  ; RK_03 电芯上料机械手压紧气缸缩回[Pls]
ANDNOT 100.06  ; RK_03 电芯上料机械手压紧气缸伸出
OUT 600.06  ; RK_03 电芯上料机械手压紧气缸伸出[A]
LD TR0
AND D1026.09  ; RK_03 电芯上料机构上料压紧气缸松开（步）
OUT 500.07  ; RK_03 电芯上料机械手压紧气缸缩回条件
TIMX(550) 0107 D18  ; 自动运行条件延时时间, RK_03 电芯上料机械手压紧气缸缩回延时[A]
LD TR0
LD 500.07  ; RK_03 电芯上料机械手压紧气缸缩回条件
AND T0107  ; RK_03 电芯上料机械手压紧气缸缩回延时[A]
OR 600.07  ; RK_03 电芯上料机械手压紧气缸缩回[A]
ANDLD
ANDNOT 500.06  ; RK_03 电芯上料机械手压紧气缸伸出条件
ANDNOT 300.07  ; RK_03 电芯上料机械手压紧气缸缩回[Pls]
ANDNOT 300.06  ; RK_03 电芯上料机械手压紧气缸伸出[Pls]
LDNOT 800.06  ; RK_03 电芯上料机械手#1压紧气缸松开位标志[0000.06]
ORNOT 800.07  ; RK_03 电芯上料机械手#2压紧气缸松开位标志[0000.07]
ANDLD
OUT 600.07  ; RK_03 电芯上料机械手压紧气缸缩回[A]

